	{attribute 'TcIecLibraryType'}
	{attribute 'external_name' := 'F_VN_InsertIntoContainer_TcVnRotatedRectangle_GUID_7CAC9217_ADAF_D1DF_8A4B_C5D37D5C5790'}
	(* Insert an element of type TcVnRotatedRectangle into a container before the specified position. *)
	FUNCTION F_VN_InsertIntoContainer_TcVnRotatedRectangle : HRESULT
	VAR_IN_OUT
		stElement	:	TcVnRotatedRectangle;	(* Single element to insert into ipContainer *)
	END_VAR
	VAR_INPUT
		ipContainer	:	ITcVnContainer;	(* Container in which to insert the element *)
		nIndex	:	ULINT;	(* Position, before which the element will be inserted *)
		hrPrev	:	HRESULT;	(* HRESULT indicating the result of previous operations (If SUCCEEDED(hrPrev) equals false, no operation is executed.) *)
	END_VAR

END_FUNCTION

// Functions/Basic Container Operations/F_VN_InsertIntoContainer/F_VN_InsertIntoContainer_TcVnVector2_DINT

	{attribute 'TcIecLibraryType'}
	{attribute 'external_name' := 'F_VN_InsertIntoContainer_TcVnVector2_DINT_GUID_6566CC88_DAB0_D931_BB59_6B341F06AF09'}
	(* Insert an element of type TcVnVector2_DINT into a container before the specified position. *)
	FUNCTION F_VN_InsertIntoContainer_TcVnVector2_DINT : HRESULT
	VAR_IN_OUT
		aElement	:	TcVnVector2_DINT;	(* Single element to insert into ipContainer *)
	END_VAR
	VAR_INPUT
		ipContainer	:	ITcVnContainer;	(* Container in which to insert the element *)
		nIndex	:	ULINT;	(* Position, before which the element will be inserted *)
		hrPrev	:	HRESULT;	(* HRESULT indicating the result of previous operations (If SUCCEEDED(hrPrev) equals false, no operation is executed.) *)
	END_VAR

END_FUNCTION

// Functions/Basic Container Operations/F_VN_InsertIntoContainer/F_VN_InsertIntoContainer_TcVnVector2_INT

	{attribute 'TcIecLibraryType'}
	{attribute 'external_name' := 'F_VN_InsertIntoContainer_TcVnVector2_INT_GUID_1A44D456_0A40_D7BF_84B8_D447168CEA63'}
	(* Insert an element of type TcVnVector2_INT into a container before the specified position. *)
	FUNCTION F_VN_InsertIntoContainer_TcVnVector2_INT : HRESULT
	VAR_IN_OUT
		aElement	:	TcVnVector2_INT;	(* Single element to insert into ipContainer *)
	END_VAR
	VAR_INPUT
		ipContainer	:	ITcVnContainer;	(* Container in which to insert the element *)
		nIndex	:	ULINT;	(* Position, before which the element will be inserted *)
		hrPrev	:	HRESULT;	(* HRESULT indicating the result of previous operations (If SUCCEEDED(hrPrev) equals false, no operation is executed.) *)
	END_VAR

END_FUNCTION

// Functions/Basic Container Operations/F_VN_InsertIntoContainer/F_VN_InsertIntoContainer_TcVnVector2_REAL

	{attribute 'TcIecLibraryType'}
	{attribute 'external_name' := 'F_VN_InsertIntoContainer_TcVnVector2_REAL_GUID_14F4E4FE_449B_DEBB_AC09_B5A9FB146C7C'}
	(* Insert an element of type TcVnVector2_REAL into a container before the specified position. *)
	FUNCTION F_VN_InsertIntoContainer_TcVnVector2_REAL : HRESULT
	VAR_IN_OUT
		aElement	:	TcVnVector2_REAL;	(* Single element to insert into ipContainer *)
	END_VAR
	VAR_INPUT
		ipContainer	:	ITcVnContainer;	(* Container in which to insert the element *)
		nIndex	:	ULINT;	(* Position, before which the element will be inserted *)
		hrPrev	:	HRESULT;	(* HRESULT indicating the result of previous operations (If SUCCEEDED(hrPrev) equals false, no operation is executed.) *)
	END_VAR

END_FUNCTION

// Functions/Basic Container Operations/F_VN_InsertIntoContainer/F_VN_InsertIntoContainer_TcVnVector2_SINT

	{attribute 'TcIecLibraryType'}
	{attribute 'external_name' := 'F_VN_InsertIntoContainer_TcVnVector2_SINT_GUID_4FA6BDE4_FC4B_D14F_9AAD_DECDAC1A2485'}
	(* Insert an element of type TcVnVector2_SINT into a container before the specified position. *)
	FUNCTION F_VN_InsertIntoContainer_TcVnVector2_SINT : HRESULT
	VAR_IN_OUT
		aElement	:	TcVnVector2_SINT;	(* Single element to insert into ipContainer *)
	END_VAR
	VAR_INPUT
		ipContainer	:	ITcVnContainer;	(* Container in which to insert the element *)
		nIndex	:	ULINT;	(* Position, before which the element will be inserted *)
		hrPrev	:	HRESULT;	(* HRESULT indicating the result of previous operations (If SUCCEEDED(hrPrev) equals false, no operation is executed.) *)
	END_VAR

END_FUNCTION

// Functions/Basic Container Operations/F_VN_InsertIntoContainer/F_VN_InsertIntoContainer_TcVnVector2_UINT

	{attribute 'TcIecLibraryType'}
	{attribute 'external_name' := 'F_VN_InsertIntoContainer_TcVnVector2_UINT_GUID_EB7FA824_1233_DA1F_B08D_37FDC60F70A2'}
	(* Insert an element of type TcVnVector2_UINT into a container before the specified position. *)
	FUNCTION F_VN_InsertIntoContainer_TcVnVector2_UINT : HRESULT
	VAR_IN_OUT
		aElement	:	TcVnVector2_UINT;	(* Single element to insert into ipContainer *)
	END_VAR
	VAR_INPUT
		ipContainer	:	ITcVnContainer;	(* Container in which to insert the element *)
		nIndex	:	ULINT;	(* Position, before which the element will be inserted *)
		hrPrev	:	HRESULT;	(* HRESULT indicating the result of previous operations (If SUCCEEDED(hrPrev) equals false, no operation is executed.) *)
	END_VAR

END_FUNCTION

// Functions/Basic Container Operations/F_VN_InsertIntoContainer/F_VN_InsertIntoContainer_TcVnVector2_USINT

	{attribute 'TcIecLibraryType'}
	{attribute 'external_name' := 'F_VN_InsertIntoContainer_TcVnVector2_USINT_GUID_68AD2749_FA5E_D5AF_8F19_582165BB6F3C'}
	(* Insert an element of type TcVnVector2_USINT into a container before the specified position. *)
	FUNCTION F_VN_InsertIntoContainer_TcVnVector2_USINT : HRESULT
	VAR_IN_OUT
		aElement	:	TcVnVector2_USINT;	(* Single element to insert into ipContainer *)
	END_VAR
	VAR_INPUT
		ipContainer	:	ITcVnContainer;	(* Container in which to insert the element *)
		nIndex	:	ULINT;	(* Position, before which the element will be inserted *)
		hrPrev	:	HRESULT;	(* HRESULT indicating the result of previous operations (If SUCCEEDED(hrPrev) equals false, no operation is executed.) *)
	END_VAR

END_FUNCTION

// Functions/Basic Container Operations/F_VN_InsertIntoContainer/F_VN_InsertIntoContainer_TcVnVector3_INT

	{attribute 'TcIecLibraryType'}
	{attribute 'external_name' := 'F_VN_InsertIntoContainer_TcVnVector3_INT_GUID_A6543EEA_C009_D51F_BEE7_FF579A0CBCDE'}
	(* Insert an element of type TcVnVector3_INT into a container before the specified position. *)
	FUNCTION F_VN_InsertIntoContainer_TcVnVector3_INT : HRESULT
	VAR_IN_OUT
		aElement	:	TcVnVector3_INT;	(* Single element to insert into ipContainer *)
	END_VAR
	VAR_INPUT
		ipContainer	:	ITcVnContainer;	(* Container in which to insert the element *)
		nIndex	:	ULINT;	(* Position, before which the element will be inserted *)
		hrPrev	:	HRESULT;	(* HRESULT indicating the result of previous operations (If SUCCEEDED(hrPrev) equals false, no operation is executed.) *)
	END_VAR

END_FUNCTION

// Functions/Basic Container Operations/F_VN_InsertIntoContainer/F_VN_InsertIntoContainer_TcVnVector3_REAL

	{attribute 'TcIecLibraryType'}
	{attribute 'external_name' := 'F_VN_InsertIntoContainer_TcVnVector3_REAL_GUID_8DA4CB93_E662_DD0B_B77C_47E33715929C'}
	(* Insert an element of type TcVnVector3_REAL into a container before the specified position. *)
	FUNCTION F_VN_InsertIntoContainer_TcVnVector3_REAL : HRESULT
	VAR_IN_OUT
		aElement	:	TcVnVector3_REAL;	(* Single element to insert into ipContainer *)
	END_VAR
	VAR_INPUT
		ipContainer	:	ITcVnContainer;	(* Container in which to insert the element *)
		nIndex	:	ULINT;	(* Position, before which the element will be inserted *)
		hrPrev	:	HRESULT;	(* HRESULT indicating the result of previous operations (If SUCCEEDED(hrPrev) equals false, no operation is executed.) *)
	END_VAR

END_FUNCTION

// Functions/Basic Container Operations/F_VN_InsertIntoContainer/F_VN_InsertIntoContainer_TcVnVector3_SINT

	{attribute 'TcIecLibraryType'}
	{attribute 'external_name' := 'F_VN_InsertIntoContainer_TcVnVector3_SINT_GUID_9F083386_9C91_DC08_8219_0E1B3C149953'}
	(* Insert an element of type TcVnVector3_SINT into a container before the specified position. *)
	FUNCTION F_VN_InsertIntoContainer_TcVnVector3_SINT : HRESULT
	VAR_IN_OUT
		aElement	:	TcVnVector3_SINT;	(* Single element to insert into ipContainer *)
	END_VAR
	VAR_INPUT
		ipContainer	:	ITcVnContainer;	(* Container in which to insert the element *)
		nIndex	:	ULINT;	(* Position, before which the element will be inserted *)
		hrPrev	:	HRESULT;	(* HRESULT indicating the result of previous operations (If SUCCEEDED(hrPrev) equals false, no operation is executed.) *)
	END_VAR

END_FUNCTION

// Functions/Basic Container Operations/F_VN_InsertIntoContainer/F_VN_InsertIntoContainer_TcVnVector3_UINT

	{attribute 'TcIecLibraryType'}
	{attribute 'external_name' := 'F_VN_InsertIntoContainer_TcVnVector3_UINT_GUID_A8405EB2_25DD_DB35_B4DF_AFF6C48501DC'}
	(* Insert an element of type TcVnVector3_UINT into a container before the specified position. *)
	FUNCTION F_VN_InsertIntoContainer_TcVnVector3_UINT : HRESULT
	VAR_IN_OUT
		aElement	:	TcVnVector3_UINT;	(* Single element to insert into ipContainer *)
	END_VAR
	VAR_INPUT
		ipContainer	:	ITcVnContainer;	(* Container in which to insert the element *)
		nIndex	:	ULINT;	(* Position, before which the element will be inserted *)
		hrPrev	:	HRESULT;	(* HRESULT indicating the result of previous operations (If SUCCEEDED(hrPrev) equals false, no operation is executed.) *)
	END_VAR

END_FUNCTION

// Functions/Basic Container Operations/F_VN_InsertIntoContainer/F_VN_InsertIntoContainer_TcVnVector3_USINT

	{attribute 'TcIecLibraryType'}
	{attribute 'external_name' := 'F_VN_InsertIntoContainer_TcVnVector3_USINT_GUID_C1142200_49EE_D153_9630_C3BAFAFB5C22'}
	(* Insert an element of type TcVnVector3_USINT into a container before the specified position. *)
	FUNCTION F_VN_InsertIntoContainer_TcVnVector3_USINT : HRESULT
	VAR_IN_OUT
		aElement	:	TcVnVector3_USINT;	(* Single element to insert into ipContainer *)
	END_VAR
	VAR_INPUT
		ipContainer	:	ITcVnContainer;	(* Container in which to insert the element *)
		nIndex	:	ULINT;	(* Position, before which the element will be inserted *)
		hrPrev	:	HRESULT;	(* HRESULT indicating the result of previous operations (If SUCCEEDED(hrPrev) equals false, no operation is executed.) *)
	END_VAR

END_FUNCTION

// Functions/Basic Container Operations/F_VN_InsertIntoContainer/F_VN_InsertIntoContainer_TcVnVector4_DINT

	{attribute 'TcIecLibraryType'}
	{attribute 'external_name' := 'F_VN_InsertIntoContainer_TcVnVector4_DINT_GUID_B98F2330_DD6A_D95D_8783_2B0449E0CC84'}
	(* Insert an element of type TcVnVector4_DINT into a container before the specified position. *)
	FUNCTION F_VN_InsertIntoContainer_TcVnVector4_DINT : HRESULT
	VAR_IN_OUT
		aElement	:	TcVnVector4_DINT;	(* Single element to insert into ipContainer *)
	END_VAR
	VAR_INPUT
		ipContainer	:	ITcVnContainer;	(* Container in which to insert the element *)
		nIndex	:	ULINT;	(* Position, before which the element will be inserted *)
		hrPrev	:	HRESULT;	(* HRESULT indicating the result of previous operations (If SUCCEEDED(hrPrev) equals false, no operation is executed.) *)
	END_VAR

END_FUNCTION

// Functions/Basic Container Operations/F_VN_InsertIntoContainer/F_VN_InsertIntoContainer_TcVnVector4_INT

	{attribute 'TcIecLibraryType'}
	{attribute 'external_name' := 'F_VN_InsertIntoContainer_TcVnVector4_INT_GUID_65611BB7_30D8_D8ED_8ECE_E86DF68481D6'}
	(* Insert an element of type TcVnVector4_INT into a container before the specified position. *)
	FUNCTION F_VN_InsertIntoContainer_TcVnVector4_INT : HRESULT
	VAR_IN_OUT
		aElement	:	TcVnVector4_INT;	(* Single element to insert into ipContainer *)
	END_VAR
	VAR_INPUT
		ipContainer	:	ITcVnContainer;	(* Container in which to insert the element *)
		nIndex	:	ULINT;	(* Position, before which the element will be inserted *)
		hrPrev	:	HRESULT;	(* HRESULT indicating the result of previous operations (If SUCCEEDED(hrPrev) equals false, no operation is executed.) *)
	END_VAR

END_FUNCTION

// Functions/Basic Container Operations/F_VN_InsertIntoContainer/F_VN_InsertIntoContainer_TcVnVector4_LREAL

	{attribute 'TcIecLibraryType'}
	{attribute 'external_name' := 'F_VN_InsertIntoContainer_TcVnVector4_LREAL_GUID_FE564EF4_0166_DE95_B96B_4103EC79B71E'}
	(* Insert an element of type TcVnVector4_LREAL into a container before the specified position. *)
	FUNCTION F_VN_InsertIntoContainer_TcVnVector4_LREAL : HRESULT
	VAR_IN_OUT
		aElement	:	TcVnVector4_LREAL;	(* Single element to insert into ipContainer *)
	END_VAR
	VAR_INPUT
		ipContainer	:	ITcVnContainer;	(* Container in which to insert the element *)
		nIndex	:	ULINT;	(* Position, before which the element will be inserted *)
		hrPrev	:	HRESULT;	(* HRESULT indicating the result of previous operations (If SUCCEEDED(hrPrev) equals false, no operation is executed.) *)
	END_VAR

END_FUNCTION

// Functions/Basic Container Operations/F_VN_InsertIntoContainer/F_VN_InsertIntoContainer_TcVnVector4_REAL

	{attribute 'TcIecLibraryType'}
	{attribute 'external_name' := 'F_VN_InsertIntoContainer_TcVnVector4_REAL_GUID_58C4540D_8F55_DF4C_9020_215109A1688E'}
	(* Insert an element of type TcVnVector4_REAL into a container before the specified position. *)
	FUNCTION F_VN_InsertIntoContainer_TcVnVector4_REAL : HRESULT
	VAR_IN_OUT
		aElement	:	TcVnVector4_REAL;	(* Single element to insert into ipContainer *)
	END_VAR
	VAR_INPUT
		ipContainer	:	ITcVnContainer;	(* Container in which to insert the element *)
		nIndex	:	ULINT;	(* Position, before which the element will be inserted *)
		hrPrev	:	HRESULT;	(* HRESULT indicating the result of previous operations (If SUCCEEDED(hrPrev) equals false, no operation is executed.) *)
	END_VAR

END_FUNCTION

// Functions/Basic Container Operations/F_VN_InsertIntoContainer/F_VN_InsertIntoContainer_TcVnVector4_SINT

	{attribute 'TcIecLibraryType'}
	{attribute 'external_name' := 'F_VN_InsertIntoContainer_TcVnVector4_SINT_GUID_E59FA623_EBB2_DB93_9AF8_202896EF00E4'}
	(* Insert an element of type TcVnVector4_SINT into a container before the specified position. *)
	FUNCTION F_VN_InsertIntoContainer_TcVnVector4_SINT : HRESULT
	VAR_IN_OUT
		aElement	:	TcVnVector4_SINT;	(* Single element to insert into ipContainer *)
	END_VAR
	VAR_INPUT
		ipContainer	:	ITcVnContainer;	(* Container in which to insert the element *)
		nIndex	:	ULINT;	(* Position, before which the element will be inserted *)
		hrPrev	:	HRESULT;	(* HRESULT indicating the result of previous operations (If SUCCEEDED(hrPrev) equals false, no operation is executed.) *)
	END_VAR

END_FUNCTION

// Functions/Basic Container Operations/F_VN_InsertIntoContainer/F_VN_InsertIntoContainer_TcVnVector4_UINT

	{attribute 'TcIecLibraryType'}
	{attribute 'external_name' := 'F_VN_InsertIntoContainer_TcVnVector4_UINT_GUID_52ADF8A2_FEB4_DF8A_9994_E3F816D9D014'}
	(* Insert an element of type TcVnVector4_UINT into a container before the specified position. *)
	FUNCTION F_VN_InsertIntoContainer_TcVnVector4_UINT : HRESULT
	VAR_IN_OUT
		aElement	:	TcVnVector4_UINT;	(* Single element to insert into ipContainer *)
	END_VAR
	VAR_INPUT
		ipContainer	:	ITcVnContainer;	(* Container in which to insert the element *)
		nIndex	:	ULINT;	(* Position, before which the element will be inserted *)
		hrPrev	:	HRESULT;	(* HRESULT indicating the result of previous operations (If SUCCEEDED(hrPrev) equals false, no operation is executed.) *)
	END_VAR

END_FUNCTION

// Functions/Basic Container Operations/F_VN_InsertIntoContainer/F_VN_InsertIntoContainer_TcVnVector4_USINT

	{attribute 'TcIecLibraryType'}
	{attribute 'external_name' := 'F_VN_InsertIntoContainer_TcVnVector4_USINT_GUID_8D180FCF_4F7F_D25B_9D06_29434C4138AE'}
	(* Insert an element of type TcVnVector4_USINT into a container before the specified position. *)
	FUNCTION F_VN_InsertIntoContainer_TcVnVector4_USINT : HRESULT
	VAR_IN_OUT
		aElement	:	TcVnVector4_USINT;	(* Single element to insert into ipContainer *)
	END_VAR
	VAR_INPUT
		ipContainer	:	ITcVnContainer;	(* Container in which to insert the element *)
		nIndex	:	ULINT;	(* Position, before which the element will be inserted *)
		hrPrev	:	HRESULT;	(* HRESULT indicating the result of previous operations (If SUCCEEDED(hrPrev) equals false, no operation is executed.) *)
	END_VAR

END_FUNCTION

// Functions/Basic Container Operations/F_VN_InsertIntoContainer/F_VN_InsertIntoContainer_UDINT

	{attribute 'TcIecLibraryType'}
	{attribute 'external_name' := 'F_VN_InsertIntoContainer_UDINT_GUID_456412AD_2528_D507_8741_196A0EE9AFE2'}
	(* Insert an element of type UDINT into a container before the specified position. *)
	FUNCTION F_VN_InsertIntoContainer_UDINT : HRESULT
	VAR_INPUT
		nElement	:	UDINT;	(* Single element to insert into ipContainer *)
		ipContainer	:	ITcVnContainer;	(* Container in which to insert the element *)
		nIndex	:	ULINT;	(* Position, before which the element will be inserted *)
		hrPrev	:	HRESULT;	(* HRESULT indicating the result of previous operations (If SUCCEEDED(hrPrev) equals false, no operation is executed.) *)
	END_VAR

END_FUNCTION

// Functions/Basic Container Operations/F_VN_InsertIntoContainer/F_VN_InsertIntoContainer_UINT

	{attribute 'TcIecLibraryType'}
	{attribute 'external_name' := 'F_VN_InsertIntoContainer_UINT_GUID_6B49D457_9F4E_DE5F_85EF_D3413FF89161'}
	(* Insert an element of type UINT into a container before the specified position. *)
	FUNCTION F_VN_InsertIntoContainer_UINT : HRESULT
	VAR_INPUT
		nElement	:	UINT;	(* Single element to insert into ipContainer *)
		ipContainer	:	ITcVnContainer;	(* Container in which to insert the element *)
		nIndex	:	ULINT;	(* Position, before which the element will be inserted *)
		hrPrev	:	HRESULT;	(* HRESULT indicating the result of previous operations (If SUCCEEDED(hrPrev) equals false, no operation is executed.) *)
	END_VAR

END_FUNCTION

// Functions/Basic Container Operations/F_VN_InsertIntoContainer/F_VN_InsertIntoContainer_ULINT

	{attribute 'TcIecLibraryType'}
	{attribute 'external_name' := 'F_VN_InsertIntoContainer_ULINT_GUID_FE1D7BC2_89AC_D4A6_855E_4E891AD80812'}
	(* Insert an element of type ULINT into a container before the specified position. *)
	FUNCTION F_VN_InsertIntoContainer_ULINT : HRESULT
	VAR_INPUT
		nElement	:	ULINT;	(* Single element to insert into ipContainer *)
		ipContainer	:	ITcVnContainer;	(* Container in which to insert the element *)
		nIndex	:	ULINT;	(* Position, before which the element will be inserted *)
		hrPrev	:	HRESULT;	(* HRESULT indicating the result of previous operations (If SUCCEEDED(hrPrev) equals false, no operation is executed.) *)
	END_VAR

END_FUNCTION

// Functions/Basic Container Operations/F_VN_InsertIntoContainer/F_VN_InsertIntoContainer_USINT

	{attribute 'TcIecLibraryType'}
	{attribute 'external_name' := 'F_VN_InsertIntoContainer_USINT_GUID_A85F087B_469C_DB69_A492_76C66B672E9A'}
	(* Insert an element of type USINT into a container before the specified position. *)
	FUNCTION F_VN_InsertIntoContainer_USINT : HRESULT
	VAR_INPUT
		nElement	:	USINT;	(* Single element to insert into ipContainer *)
		ipContainer	:	ITcVnContainer;	(* Container in which to insert the element *)
		nIndex	:	ULINT;	(* Position, before which the element will be inserted *)
		hrPrev	:	HRESULT;	(* HRESULT indicating the result of previous operations (If SUCCEEDED(hrPrev) equals false, no operation is executed.) *)
	END_VAR

END_FUNCTION

// Functions/Basic Container Operations/F_VN_SetAt/F_VN_SetAt_ITcVnContainer

	{attribute 'TcIecLibraryType'}
	{attribute 'external_name' := 'F_VN_SetAt_ITcVnContainer_GUID_B4D766E9_0AA2_DD2D_B478_52D12AAD3DA2'}
	(* Sets the element at the specified index of the container. (Alternatively use interface method .SetAt.) *)
	FUNCTION F_VN_SetAt_ITcVnContainer : HRESULT
	VAR_INPUT
		ipElement	:	ITcVnContainer;	(* Element to set at the specified container position *)
		ipContainer	:	ITcVnContainer;	(* Container with ITcVnContainer elements, in which the element at position nIndex is replaced by ipElement *)
		nIndex	:	ULINT;	(* Index *)
		hrPrev	:	HRESULT;	(* HRESULT indicating the result of previous operations (If SUCCEEDED(hrPrev) equals false, no operation is executed.) *)
	END_VAR

END_FUNCTION

// Functions/Basic Container Operations/F_VN_SetAt/F_VN_SetAt_DINT

	{attribute 'TcIecLibraryType'}
	{attribute 'external_name' := 'F_VN_SetAt_DINT_GUID_253433CB_2425_DDF0_8BE6_B05C6CBF2EB5'}
	(* Sets the element at the specified index of the container. *)
	FUNCTION F_VN_SetAt_DINT : HRESULT
	VAR_INPUT
		nElement	:	DINT;	(* Element to set at the specified container position *)
		ipContainer	:	ITcVnContainer;	(* Container with DINT elements, in which the element at position nIndex is replaced by nElement *)
		nIndex	:	ULINT;	(* Index *)
		hrPrev	:	HRESULT;	(* HRESULT indicating the result of previous operations (If SUCCEEDED(hrPrev) equals false, no operation is executed.) *)
	END_VAR

END_FUNCTION

// Functions/Basic Container Operations/F_VN_SetAt/F_VN_SetAt_INT

	{attribute 'TcIecLibraryType'}
	{attribute 'external_name' := 'F_VN_SetAt_INT_GUID_B0E2F6D5_1415_D22F_A65C_C36499F3DF8D'}
	(* Sets the element at the specified index of the container. *)
	FUNCTION F_VN_SetAt_INT : HRESULT
	VAR_INPUT
		nElement	:	INT;	(* Element to set at the specified container position *)
		ipContainer	:	ITcVnContainer;	(* Container with INT elements, in which the element at position nIndex is replaced by nElement *)
		nIndex	:	ULINT;	(* Index *)
		hrPrev	:	HRESULT;	(* HRESULT indicating the result of previous operations (If SUCCEEDED(hrPrev) equals false, no operation is executed.) *)
	END_VAR

END_FUNCTION

// Functions/Basic Container Operations/F_VN_SetAt/F_VN_SetAt_ITcVnImage

	{attribute 'TcIecLibraryType'}
	{attribute 'external_name' := 'F_VN_SetAt_ITcVnImage_GUID_8BFD8EA5_9C85_DADE_A61A_698800738790'}
	(* Sets the element at the specified index of the container. *)
	FUNCTION F_VN_SetAt_ITcVnImage : HRESULT
	VAR_INPUT
		ipElement	:	ITcVnImage;	(* Element to set at the specified container position *)
		ipContainer	:	ITcVnContainer;	(* Container with ITcVnImage elements, in which the element at position nIndex is replaced by ipElement *)
		nIndex	:	ULINT;	(* Index *)
		hrPrev	:	HRESULT;	(* HRESULT indicating the result of previous operations (If SUCCEEDED(hrPrev) equals false, no operation is executed.) *)
	END_VAR

END_FUNCTION

// Functions/Basic Container Operations/F_VN_SetAt/F_VN_SetAt_LREAL

	{attribute 'TcIecLibraryType'}
	{attribute 'external_name' := 'F_VN_SetAt_LREAL_GUID_B183A29F_8335_D912_8808_5352ACF3B9D5'}
	(* Sets the element at the specified index of the container. *)
	FUNCTION F_VN_SetAt_LREAL : HRESULT
	VAR_INPUT
		fElement	:	LREAL;	(* Element to set at the specified container position *)
		ipContainer	:	ITcVnContainer;	(* Container with LREAL elements, in which the element at position nIndex is replaced by fElement *)
		nIndex	:	ULINT;	(* Index *)
		hrPrev	:	HRESULT;	(* HRESULT indicating the result of previous operations (If SUCCEEDED(hrPrev) equals false, no operation is executed.) *)
	END_VAR

END_FUNCTION

// Functions/Basic Container Operations/F_VN_SetAt/F_VN_SetAt_REAL

	{attribute 'TcIecLibraryType'}
	{attribute 'external_name' := 'F_VN_SetAt_REAL_GUID_7E957C6A_9FEC_D57C_9D71_8DD5085B7449'}
	(* Sets the element at the specified index of the container. *)
	FUNCTION F_VN_SetAt_REAL : HRESULT
	VAR_INPUT
		fElement	:	REAL;	(* Element to set at the specified container position *)
		ipContainer	:	ITcVnContainer;	(* Container with REAL elements, in which the element at position nIndex is replaced by fElement *)
		nIndex	:	ULINT;	(* Index *)
		hrPrev	:	HRESULT;	(* HRESULT indicating the result of previous operations (If SUCCEEDED(hrPrev) equals false, no operation is executed.) *)
	END_VAR

END_FUNCTION

// Functions/Basic Container Operations/F_VN_SetAt/F_VN_SetAt_SINT

	{attribute 'TcIecLibraryType'}
	{attribute 'external_name' := 'F_VN_SetAt_SINT_GUID_A0498278_0B8F_D4D0_B592_136B0477C0F3'}
	(* Sets the element at the specified index of the container. *)
	FUNCTION F_VN_SetAt_SINT : HRESULT
	VAR_INPUT
		nElement	:	SINT;	(* Element to set at the specified container position *)
		ipContainer	:	ITcVnContainer;	(* Container with SINT elements, in which the element at position nIndex is replaced by nElement *)
		nIndex	:	ULINT;	(* Index *)
		hrPrev	:	HRESULT;	(* HRESULT indicating the result of previous operations (If SUCCEEDED(hrPrev) equals false, no operation is executed.) *)
	END_VAR

END_FUNCTION

// Functions/Basic Container Operations/F_VN_SetAt/F_VN_SetAt_TcVnDMatch

	{attribute 'TcIecLibraryType'}
	{attribute 'external_name' := 'F_VN_SetAt_TcVnDMatch_GUID_2DD68088_896B_D3C6_AD71_4673DA0389D4'}
	(* Sets the element at the specified index of the container. *)
	FUNCTION F_VN_SetAt_TcVnDMatch : HRESULT
	VAR_IN_OUT
		stElement	:	TcVnDMatch;	(* Element to set at the specified container position *)
	END_VAR
	VAR_INPUT
		ipContainer	:	ITcVnContainer;	(* Container with TcVnDMatch elements, in which the element at position nIndex is replaced by stElement *)
		nIndex	:	ULINT;	(* Index *)
		hrPrev	:	HRESULT;	(* HRESULT indicating the result of previous operations (If SUCCEEDED(hrPrev) equals false, no operation is executed.) *)
	END_VAR

END_FUNCTION

// Functions/Basic Container Operations/F_VN_SetAt/F_VN_SetAt_TcVnKeyPoint

	{attribute 'TcIecLibraryType'}
	{attribute 'external_name' := 'F_VN_SetAt_TcVnKeyPoint_GUID_5542B220_7839_DF8E_B6D3_14C96E222448'}
	(* Sets the element at the specified index of the container. *)
	FUNCTION F_VN_SetAt_TcVnKeyPoint : HRESULT
	VAR_IN_OUT
		stElement	:	TcVnKeyPoint;	(* Element to set at the specified container position *)
	END_VAR
	VAR_INPUT
		ipContainer	:	ITcVnContainer;	(* Container with TcVnKeyPoint elements, in which the element at position nIndex is replaced by stElement *)
		nIndex	:	ULINT;	(* Index *)
		hrPrev	:	HRESULT;	(* HRESULT indicating the result of previous operations (If SUCCEEDED(hrPrev) equals false, no operation is executed.) *)
	END_VAR

END_FUNCTION

// Functions/Basic Container Operations/F_VN_SetAt/F_VN_SetAt_TcVnPoint2_DINT

	{attribute 'TcIecLibraryType'}
	{attribute 'external_name' := 'F_VN_SetAt_TcVnPoint2_DINT_GUID_380C3A28_A538_D35A_886E_4DB239484DC0'}
	(* Sets the element at the specified index of the container. *)
	FUNCTION F_VN_SetAt_TcVnPoint2_DINT : HRESULT
	VAR_IN_OUT
		aElement	:	TcVnPoint2_DINT;	(* Element to set at the specified container position *)
	END_VAR
	VAR_INPUT
		ipContainer	:	ITcVnContainer;	(* Container with TcVnPoint2_DINT elements, in which the element at position nIndex is replaced by aElement *)
		nIndex	:	ULINT;	(* Index *)
		hrPrev	:	HRESULT;	(* HRESULT indicating the result of previous operations (If SUCCEEDED(hrPrev) equals false, no operation is executed.) *)
	END_VAR

END_FUNCTION

// Functions/Basic Container Operations/F_VN_SetAt/F_VN_SetAt_TcVnPoint2_LREAL

	{attribute 'TcIecLibraryType'}
	{attribute 'external_name' := 'F_VN_SetAt_TcVnPoint2_LREAL_GUID_3335CF1D_E3D4_D03B_9014_F1A43D08A30F'}
	(* Sets the element at the specified index of the container. *)
	FUNCTION F_VN_SetAt_TcVnPoint2_LREAL : HRESULT
	VAR_IN_OUT
		aElement	:	TcVnPoint2_LREAL;	(* Element to set at the specified container position *)
	END_VAR
	VAR_INPUT
		ipContainer	:	ITcVnContainer;	(* Container with TcVnPoint2_LREAL elements, in which the element at position nIndex is replaced by aElement *)
		nIndex	:	ULINT;	(* Index *)
		hrPrev	:	HRESULT;	(* HRESULT indicating the result of previous operations (If SUCCEEDED(hrPrev) equals false, no operation is executed.) *)
	END_VAR

END_FUNCTION

// Functions/Basic Container Operations/F_VN_SetAt/F_VN_SetAt_TcVnPoint2_REAL

	{attribute 'TcIecLibraryType'}
	{attribute 'external_name' := 'F_VN_SetAt_TcVnPoint2_REAL_GUID_633C5783_5133_DC7E_ABCC_93BD16D56EFF'}
	(* Sets the element at the specified index of the container. *)
	FUNCTION F_VN_SetAt_TcVnPoint2_REAL : HRESULT
	VAR_IN_OUT
		aElement	:	TcVnPoint2_REAL;	(* Element to set at the specified container position *)
	END_VAR
	VAR_INPUT
		ipContainer	:	ITcVnContainer;	(* Container with TcVnPoint2_REAL elements, in which the element at position nIndex is replaced by aElement *)
		nIndex	:	ULINT;	(* Index *)
		hrPrev	:	HRESULT;	(* HRESULT indicating the result of previous operations (If SUCCEEDED(hrPrev) equals false, no operation is executed.) *)
	END_VAR

END_FUNCTION

// Functions/Basic Container Operations/F_VN_SetAt/F_VN_SetAt_TcVnPoint3_LREAL

	{attribute 'TcIecLibraryType'}
	{attribute 'external_name' := 'F_VN_SetAt_TcVnPoint3_LREAL_GUID_FA067292_14A4_D164_A359_A281C2761513'}
	(* Sets the element at the specified index of the container. *)
	FUNCTION F_VN_SetAt_TcVnPoint3_LREAL : HRESULT
	VAR_IN_OUT
		aElement	:	TcVnPoint3_LREAL;	(* Element to set at the specified container position *)
	END_VAR
	VAR_INPUT
		ipContainer	:	ITcVnContainer;	(* Container with TcVnPoint3_LREAL elements, in which the element at position nIndex is replaced by aElement *)
		nIndex	:	ULINT;	(* Index *)
		hrPrev	:	HRESULT;	(* HRESULT indicating the result of previous operations (If SUCCEEDED(hrPrev) equals false, no operation is executed.) *)
	END_VAR

END_FUNCTION

// Functions/Basic Container Operations/F_VN_SetAt/F_VN_SetAt_TcVnPoint3_REAL

	{attribute 'TcIecLibraryType'}
	{attribute 'external_name' := 'F_VN_SetAt_TcVnPoint3_REAL_GUID_C913190D_69EF_DE67_9951_6D3EB8AF0AD3'}
	(* Sets the element at the specified index of the container. *)
	FUNCTION F_VN_SetAt_TcVnPoint3_REAL : HRESULT
	VAR_IN_OUT
		aElement	:	TcVnPoint3_REAL;	(* Element to set at the specified container position *)
	END_VAR
	VAR_INPUT
		ipContainer	:	ITcVnContainer;	(* Container with TcVnPoint3_REAL elements, in which the element at position nIndex is replaced by aElement *)
		nIndex	:	ULINT;	(* Index *)
		hrPrev	:	HRESULT;	(* HRESULT indicating the result of previous operations (If SUCCEEDED(hrPrev) equals false, no operation is executed.) *)
	END_VAR

END_FUNCTION

// Functions/Basic Container Operations/F_VN_SetAt/F_VN_SetAt_TcVnRectangle_DINT

	{attribute 'TcIecLibraryType'}
	{attribute 'external_name' := 'F_VN_SetAt_TcVnRectangle_DINT_GUID_4532A8D1_EA7C_DA26_B932_400B95600032'}
	(* Sets the element at the specified index of the container. *)
	FUNCTION F_VN_SetAt_TcVnRectangle_DINT : HRESULT
	VAR_IN_OUT
		stElement	:	TcVnRectangle_DINT;	(* Element to set at the specified container position *)
	END_VAR
	VAR_INPUT
		ipContainer	:	ITcVnContainer;	(* Container with TcVnRectangle_DINT elements, in which the element at position nIndex is replaced by stElement *)
		nIndex	:	ULINT;	(* Index *)
		hrPrev	:	HRESULT;	(* HRESULT indicating the result of previous operations (If SUCCEEDED(hrPrev) equals false, no operation is executed.) *)
	END_VAR

END_FUNCTION

// Functions/Basic Container Operations/F_VN_SetAt/F_VN_SetAt_TcVnRotatedRectangle

	{attribute 'TcIecLibraryType'}
	{attribute 'external_name' := 'F_VN_SetAt_TcVnRotatedRectangle_GUID_DAFC69FA_D3C4_DF12_83F3_1F7CE1D06A87'}
	(* Sets the element at the specified index of the container. *)
	FUNCTION F_VN_SetAt_TcVnRotatedRectangle : HRESULT
	VAR_IN_OUT
		stElement	:	TcVnRotatedRectangle;	(* Element to set at the specified container position *)
	END_VAR
	VAR_INPUT
		ipContainer	:	ITcVnContainer;	(* Container with TcVnRotatedRectangle elements, in which the element at position nIndex is replaced by stElement *)
		nIndex	:	ULINT;	(* Index *)
		hrPrev	:	HRESULT;	(* HRESULT indicating the result of previous operations (If SUCCEEDED(hrPrev) equals false, no operation is executed.) *)
	END_VAR

END_FUNCTION

// Functions/Basic Container Operations/F_VN_SetAt/F_VN_SetAt_TcVnVector2_DINT

	{attribute 'TcIecLibraryType'}
	{attribute 'external_name' := 'F_VN_SetAt_TcVnVector2_DINT_GUID_2E9C4D9D_A279_D002_86E8_DAA9F02A0E05'}
	(* Sets the element at the specified index of the container. *)
	FUNCTION F_VN_SetAt_TcVnVector2_DINT : HRESULT
	VAR_IN_OUT
		aElement	:	TcVnVector2_DINT;	(* Element to set at the specified container position *)
	END_VAR
	VAR_INPUT
		ipContainer	:	ITcVnContainer;	(* Container with TcVnVector2_DINT elements, in which the element at position nIndex is replaced by aElement *)
		nIndex	:	ULINT;	(* Index *)
		hrPrev	:	HRESULT;	(* HRESULT indicating the result of previous operations (If SUCCEEDED(hrPrev) equals false, no operation is executed.) *)
	END_VAR

END_FUNCTION

// Functions/Basic Container Operations/F_VN_SetAt/F_VN_SetAt_TcVnVector2_INT

	{attribute 'TcIecLibraryType'}
	{attribute 'external_name' := 'F_VN_SetAt_TcVnVector2_INT_GUID_EACA2057_16BA_D239_9B9E_74E17D255685'}
	(* Sets the element at the specified index of the container. *)
	FUNCTION F_VN_SetAt_TcVnVector2_INT : HRESULT
	VAR_IN_OUT
		aElement	:	TcVnVector2_INT;	(* Element to set at the specified container position *)
	END_VAR
	VAR_INPUT
		ipContainer	:	ITcVnContainer;	(* Container with TcVnVector2_INT elements, in which the element at position nIndex is replaced by aElement *)
		nIndex	:	ULINT;	(* Index *)
		hrPrev	:	HRESULT;	(* HRESULT indicating the result of previous operations (If SUCCEEDED(hrPrev) equals false, no operation is executed.) *)
	END_VAR

END_FUNCTION

// Functions/Basic Container Operations/F_VN_SetAt/F_VN_SetAt_TcVnVector2_REAL

	{attribute 'TcIecLibraryType'}
	{attribute 'external_name' := 'F_VN_SetAt_TcVnVector2_REAL_GUID_FCEEF9F1_A95E_D6B4_82C2_0524AF8ED162'}
	(* Sets the element at the specified index of the container. *)
	FUNCTION F_VN_SetAt_TcVnVector2_REAL : HRESULT
	VAR_IN_OUT
		aElement	:	TcVnVector2_REAL;	(* Element to set at the specified container position *)
	END_VAR
	VAR_INPUT
		ipContainer	:	ITcVnContainer;	(* Container with TcVnVector2_REAL elements, in which the element at position nIndex is replaced by aElement *)
		nIndex	:	ULINT;	(* Index *)
		hrPrev	:	HRESULT;	(* HRESULT indicating the result of previous operations (If SUCCEEDED(hrPrev) equals false, no operation is executed.) *)
	END_VAR

END_FUNCTION

// Functions/Basic Container Operations/F_VN_SetAt/F_VN_SetAt_TcVnVector2_SINT

	{attribute 'TcIecLibraryType'}
	{attribute 'external_name' := 'F_VN_SetAt_TcVnVector2_SINT_GUID_317C493E_1B6C_DEE3_AE25_CC2C29021A66'}
	(* Sets the element at the specified index of the container. *)
	FUNCTION F_VN_SetAt_TcVnVector2_SINT : HRESULT
	VAR_IN_OUT
		aElement	:	TcVnVector2_SINT;	(* Element to set at the specified container position *)
	END_VAR
	VAR_INPUT
		ipContainer	:	ITcVnContainer;	(* Container with TcVnVector2_SINT elements, in which the element at position nIndex is replaced by aElement *)
		nIndex	:	ULINT;	(* Index *)
		hrPrev	:	HRESULT;	(* HRESULT indicating the result of previous operations (If SUCCEEDED(hrPrev) equals false, no operation is executed.) *)
	END_VAR

END_FUNCTION

// Functions/Basic Container Operations/F_VN_SetAt/F_VN_SetAt_TcVnVector2_UINT

	{attribute 'TcIecLibraryType'}
	{attribute 'external_name' := 'F_VN_SetAt_TcVnVector2_UINT_GUID_51607B5B_B463_D36D_8B37_1F9AE2FB26C1'}
	(* Sets the element at the specified index of the container. *)
	FUNCTION F_VN_SetAt_TcVnVector2_UINT : HRESULT
	VAR_IN_OUT
		aElement	:	TcVnVector2_UINT;	(* Element to set at the specified container position *)
	END_VAR
	VAR_INPUT
		ipContainer	:	ITcVnContainer;	(* Container with TcVnVector2_UINT elements, in which the element at position nIndex is replaced by aElement *)
		nIndex	:	ULINT;	(* Index *)
		hrPrev	:	HRESULT;	(* HRESULT indicating the result of previous operations (If SUCCEEDED(hrPrev) equals false, no operation is executed.) *)
	END_VAR

END_FUNCTION

// Functions/Basic Container Operations/F_VN_SetAt/F_VN_SetAt_TcVnVector2_USINT

	{attribute 'TcIecLibraryType'}
	{attribute 'external_name' := 'F_VN_SetAt_TcVnVector2_USINT_GUID_01F9C5AE_E454_D0D0_90FA_2E0A2E622C7C'}
	(* Sets the element at the specified index of the container. *)
	FUNCTION F_VN_SetAt_TcVnVector2_USINT : HRESULT
	VAR_IN_OUT
		aElement	:	TcVnVector2_USINT;	(* Element to set at the specified container position *)
	END_VAR
	VAR_INPUT
		ipContainer	:	ITcVnContainer;	(* Container with TcVnVector2_USINT elements, in which the element at position nIndex is replaced by aElement *)
		nIndex	:	ULINT;	(* Index *)
		hrPrev	:	HRESULT;	(* HRESULT indicating the result of previous operations (If SUCCEEDED(hrPrev) equals false, no operation is executed.) *)
	END_VAR

END_FUNCTION

// Functions/Basic Container Operations/F_VN_SetAt/F_VN_SetAt_TcVnVector3_INT

	{attribute 'TcIecLibraryType'}
	{attribute 'external_name' := 'F_VN_SetAt_TcVnVector3_INT_GUID_C31915F3_E342_D7E4_A41C_3483F9896BDE'}
	(* Sets the element at the specified index of the container. *)
	FUNCTION F_VN_SetAt_TcVnVector3_INT : HRESULT
	VAR_IN_OUT
		aElement	:	TcVnVector3_INT;	(* Element to set at the specified container position *)
	END_VAR
	VAR_INPUT
		ipContainer	:	ITcVnContainer;	(* Container with TcVnVector3_INT elements, in which the element at position nIndex is replaced by aElement *)
		nIndex	:	ULINT;	(* Index *)
		hrPrev	:	HRESULT;	(* HRESULT indicating the result of previous operations (If SUCCEEDED(hrPrev) equals false, no operation is executed.) *)
	END_VAR

END_FUNCTION

// Functions/Basic Container Operations/F_VN_SetAt/F_VN_SetAt_TcVnVector3_REAL

	{attribute 'TcIecLibraryType'}
	{attribute 'external_name' := 'F_VN_SetAt_TcVnVector3_REAL_GUID_E7E10DE5_BBDC_D2B5_82C3_D03B676D1019'}
	(* Sets the element at the specified index of the container. *)
	FUNCTION F_VN_SetAt_TcVnVector3_REAL : HRESULT
	VAR_IN_OUT
		aElement	:	TcVnVector3_REAL;	(* Element to set at the specified container position *)
	END_VAR
	VAR_INPUT
		ipContainer	:	ITcVnContainer;	(* Container with TcVnVector3_REAL elements, in which the element at position nIndex is replaced by aElement *)
		nIndex	:	ULINT;	(* Index *)
		hrPrev	:	HRESULT;	(* HRESULT indicating the result of previous operations (If SUCCEEDED(hrPrev) equals false, no operation is executed.) *)
	END_VAR

END_FUNCTION

// Functions/Basic Container Operations/F_VN_SetAt/F_VN_SetAt_TcVnVector3_SINT

	{attribute 'TcIecLibraryType'}
	{attribute 'external_name' := 'F_VN_SetAt_TcVnVector3_SINT_GUID_F25AB548_5F5E_DC98_B6BC_12B5548547A2'}
	(* Sets the element at the specified index of the container. *)
	FUNCTION F_VN_SetAt_TcVnVector3_SINT : HRESULT
	VAR_IN_OUT
		aElement	:	TcVnVector3_SINT;	(* Element to set at the specified container position *)
	END_VAR
	VAR_INPUT
		ipContainer	:	ITcVnContainer;	(* Container with TcVnVector3_SINT elements, in which the element at position nIndex is replaced by aElement *)
		nIndex	:	ULINT;	(* Index *)
		hrPrev	:	HRESULT;	(* HRESULT indicating the result of previous operations (If SUCCEEDED(hrPrev) equals false, no operation is executed.) *)
	END_VAR

END_FUNCTION

// Functions/Basic Container Operations/F_VN_SetAt/F_VN_SetAt_TcVnVector3_UINT

	{attribute 'TcIecLibraryType'}
	{attribute 'external_name' := 'F_VN_SetAt_TcVnVector3_UINT_GUID_C0EAE934_C854_D169_9697_13D208B74332'}
	(* Sets the element at the specified index of the container. *)
	FUNCTION F_VN_SetAt_TcVnVector3_UINT : HRESULT
	VAR_IN_OUT
		aElement	:	TcVnVector3_UINT;	(* Element to set at the specified container position *)
	END_VAR
	VAR_INPUT
		ipContainer	:	ITcVnContainer;	(* Container with TcVnVector3_UINT elements, in which the element at position nIndex is replaced by aElement *)
		nIndex	:	ULINT;	(* Index *)
		hrPrev	:	HRESULT;	(* HRESULT indicating the result of previous operations (If SUCCEEDED(hrPrev) equals false, no operation is executed.) *)
	END_VAR

END_FUNCTION

// Functions/Basic Container Operations/F_VN_SetAt/F_VN_SetAt_TcVnVector3_USINT

	{attribute 'TcIecLibraryType'}
	{attribute 'external_name' := 'F_VN_SetAt_TcVnVector3_USINT_GUID_BA06F0BE_A1AF_D5B9_9020_C48B8FF58FCA'}
	(* Sets the element at the specified index of the container. *)
	FUNCTION F_VN_SetAt_TcVnVector3_USINT : HRESULT
	VAR_IN_OUT
		aElement	:	TcVnVector3_USINT;	(* Element to set at the specified container position *)
	END_VAR
	VAR_INPUT
		ipContainer	:	ITcVnContainer;	(* Container with TcVnVector3_USINT elements, in which the element at position nIndex is replaced by aElement *)
		nIndex	:	ULINT;	(* Index *)
		hrPrev	:	HRESULT;	(* HRESULT indicating the result of previous operations (If SUCCEEDED(hrPrev) equals false, no operation is executed.) *)
	END_VAR

END_FUNCTION

// Functions/Basic Container Operations/F_VN_SetAt/F_VN_SetAt_TcVnVector4_DINT

	{attribute 'TcIecLibraryType'}
	{attribute 'external_name' := 'F_VN_SetAt_TcVnVector4_DINT_GUID_F499B98D_2623_D67F_9D86_B597EF831028'}
	(* Sets the element at the specified index of the container. *)
	FUNCTION F_VN_SetAt_TcVnVector4_DINT : HRESULT
	VAR_IN_OUT
		aElement	:	TcVnVector4_DINT;	(* Element to set at the specified container position *)
	END_VAR
	VAR_INPUT
		ipContainer	:	ITcVnContainer;	(* Container with TcVnVector4_DINT elements, in which the element at position nIndex is replaced by aElement *)
		nIndex	:	ULINT;	(* Index *)
		hrPrev	:	HRESULT;	(* HRESULT indicating the result of previous operations (If SUCCEEDED(hrPrev) equals false, no operation is executed.) *)
	END_VAR

END_FUNCTION

// Functions/Basic Container Operations/F_VN_SetAt/F_VN_SetAt_TcVnVector4_INT

	{attribute 'TcIecLibraryType'}
	{attribute 'external_name' := 'F_VN_SetAt_TcVnVector4_INT_GUID_3C1822B1_48CA_DE5C_9E46_7B4DAA7D5C91'}
	(* Sets the element at the specified index of the container. *)
	FUNCTION F_VN_SetAt_TcVnVector4_INT : HRESULT
	VAR_IN_OUT
		aElement	:	TcVnVector4_INT;	(* Element to set at the specified container position *)
	END_VAR
	VAR_INPUT
		ipContainer	:	ITcVnContainer;	(* Container with TcVnVector4_INT elements, in which the element at position nIndex is replaced by aElement *)
		nIndex	:	ULINT;	(* Index *)
		hrPrev	:	HRESULT;	(* HRESULT indicating the result of previous operations (If SUCCEEDED(hrPrev) equals false, no operation is executed.) *)
	END_VAR

END_FUNCTION

// Functions/Basic Container Operations/F_VN_SetAt/F_VN_SetAt_TcVnVector4_LREAL

	{attribute 'TcIecLibraryType'}
	{attribute 'external_name' := 'F_VN_SetAt_TcVnVector4_LREAL_GUID_C31FA288_C1E2_DFBA_959D_2529D6A83E64'}
	(* Sets the element at the specified index of the container. *)
	FUNCTION F_VN_SetAt_TcVnVector4_LREAL : HRESULT
	VAR_IN_OUT
		aElement	:	TcVnVector4_LREAL;	(* Element to set at the specified container position *)
	END_VAR
	VAR_INPUT
		ipContainer	:	ITcVnContainer;	(* Container with TcVnVector4_LREAL elements, in which the element at position nIndex is replaced by aElement *)
		nIndex	:	ULINT;	(* Index *)
		hrPrev	:	HRESULT;	(* HRESULT indicating the result of previous operations (If SUCCEEDED(hrPrev) equals false, no operation is executed.) *)
	END_VAR

END_FUNCTION

// Functions/Basic Container Operations/F_VN_SetAt/F_VN_SetAt_TcVnVector4_REAL

	{attribute 'TcIecLibraryType'}
	{attribute 'external_name' := 'F_VN_SetAt_TcVnVector4_REAL_GUID_14303487_AE28_D413_B77E_42801EACBB76'}
	(* Sets the element at the specified index of the container. *)
	FUNCTION F_VN_SetAt_TcVnVector4_REAL : HRESULT
	VAR_IN_OUT
		aElement	:	TcVnVector4_REAL;	(* Element to set at the specified container position *)
	END_VAR
	VAR_INPUT
		ipContainer	:	ITcVnContainer;	(* Container with TcVnVector4_REAL elements, in which the element at position nIndex is replaced by aElement *)
		nIndex	:	ULINT;	(* Index *)
		hrPrev	:	HRESULT;	(* HRESULT indicating the result of previous operations (If SUCCEEDED(hrPrev) equals false, no operation is executed.) *)
	END_VAR

END_FUNCTION

// Functions/Basic Container Operations/F_VN_SetAt/F_VN_SetAt_TcVnVector4_SINT

	{attribute 'TcIecLibraryType'}
	{attribute 'external_name' := 'F_VN_SetAt_TcVnVector4_SINT_GUID_EABA744D_28BE_D87B_AF4B_7CA5F5619B72'}
	(* Sets the element at the specified index of the container. *)
	FUNCTION F_VN_SetAt_TcVnVector4_SINT : HRESULT
	VAR_IN_OUT
		aElement	:	TcVnVector4_SINT;	(* Element to set at the specified container position *)
	END_VAR
	VAR_INPUT
		ipContainer	:	ITcVnContainer;	(* Container with TcVnVector4_SINT elements, in which the element at position nIndex is replaced by aElement *)
		nIndex	:	ULINT;	(* Index *)
		hrPrev	:	HRESULT;	(* HRESULT indicating the result of previous operations (If SUCCEEDED(hrPrev) equals false, no operation is executed.) *)
	END_VAR

END_FUNCTION

// Functions/Basic Container Operations/F_VN_SetAt/F_VN_SetAt_TcVnVector4_UINT

	{attribute 'TcIecLibraryType'}
	{attribute 'external_name' := 'F_VN_SetAt_TcVnVector4_UINT_GUID_ECE2D899_7CF8_D3D2_B546_AEA5C3AC0E78'}
	(* Sets the element at the specified index of the container. *)
	FUNCTION F_VN_SetAt_TcVnVector4_UINT : HRESULT
	VAR_IN_OUT
		aElement	:	TcVnVector4_UINT;	(* Element to set at the specified container position *)
	END_VAR
	VAR_INPUT
		ipContainer	:	ITcVnContainer;	(* Container with TcVnVector4_UINT elements, in which the element at position nIndex is replaced by aElement *)
		nIndex	:	ULINT;	(* Index *)
		hrPrev	:	HRESULT;	(* HRESULT indicating the result of previous operations (If SUCCEEDED(hrPrev) equals false, no operation is executed.) *)
	END_VAR

END_FUNCTION

// Functions/Basic Container Operations/F_VN_SetAt/F_VN_SetAt_TcVnVector4_USINT

	{attribute 'TcIecLibraryType'}
	{attribute 'external_name' := 'F_VN_SetAt_TcVnVector4_USINT_GUID_FC552792_92A1_D187_8C56_50F5B0CDF203'}
	(* Sets the element at the specified index of the container. *)
	FUNCTION F_VN_SetAt_TcVnVector4_USINT : HRESULT
	VAR_IN_OUT
		aElement	:	TcVnVector4_USINT;	(* Element to set at the specified container position *)
	END_VAR
	VAR_INPUT
		ipContainer	:	ITcVnContainer;	(* Container with TcVnVector4_USINT elements, in which the element at position nIndex is replaced by aElement *)
		nIndex	:	ULINT;	(* Index *)
		hrPrev	:	HRESULT;	(* HRESULT indicating the result of previous operations (If SUCCEEDED(hrPrev) equals false, no operation is executed.) *)
	END_VAR

END_FUNCTION

// Functions/Basic Container Operations/F_VN_SetAt/F_VN_SetAt_UDINT

	{attribute 'TcIecLibraryType'}
	{attribute 'external_name' := 'F_VN_SetAt_UDINT_GUID_B305A6D1_2AE2_D412_9BD3_F3AF279AFF3A'}
	(* Sets the element at the specified index of the container. *)
	FUNCTION F_VN_SetAt_UDINT : HRESULT
	VAR_INPUT
		nElement	:	UDINT;	(* Element to set at the specified container position *)
		ipContainer	:	ITcVnContainer;	(* Container with UDINT elements, in which the element at position nIndex is replaced by nElement *)
		nIndex	:	ULINT;	(* Index *)
		hrPrev	:	HRESULT;	(* HRESULT indicating the result of previous operations (If SUCCEEDED(hrPrev) equals false, no operation is executed.) *)
	END_VAR

END_FUNCTION

// Functions/Basic Container Operations/F_VN_SetAt/F_VN_SetAt_UINT

	{attribute 'TcIecLibraryType'}
	{attribute 'external_name' := 'F_VN_SetAt_UINT_GUID_E7A3ED31_6DA7_DBE5_B80B_892891209441'}
	(* Sets the element at the specified index of the container. *)
	FUNCTION F_VN_SetAt_UINT : HRESULT
	VAR_INPUT
		nElement	:	UINT;	(* Element to set at the specified container position *)
		ipContainer	:	ITcVnContainer;	(* Container with UINT elements, in which the element at position nIndex is replaced by nElement *)
		nIndex	:	ULINT;	(* Index *)
		hrPrev	:	HRESULT;	(* HRESULT indicating the result of previous operations (If SUCCEEDED(hrPrev) equals false, no operation is executed.) *)
	END_VAR

END_FUNCTION

// Functions/Basic Container Operations/F_VN_SetAt/F_VN_SetAt_ULINT

	{attribute 'TcIecLibraryType'}
	{attribute 'external_name' := 'F_VN_SetAt_ULINT_GUID_8C16F2A2_3A38_D764_A670_EC92096893B4'}
	(* Sets the element at the specified index of the container. *)
	FUNCTION F_VN_SetAt_ULINT : HRESULT
	VAR_INPUT
		nElement	:	ULINT;	(* Element to set at the specified container position *)
		ipContainer	:	ITcVnContainer;	(* Container with ULINT elements, in which the element at position nIndex is replaced by nElement *)
		nIndex	:	ULINT;	(* Index *)
		hrPrev	:	HRESULT;	(* HRESULT indicating the result of previous operations (If SUCCEEDED(hrPrev) equals false, no operation is executed.) *)
	END_VAR

END_FUNCTION

// Functions/Basic Container Operations/F_VN_SetAt/F_VN_SetAt_USINT

	{attribute 'TcIecLibraryType'}
	{attribute 'external_name' := 'F_VN_SetAt_USINT_GUID_01F9B48C_F95B_D032_BABB_6175AD7802C9'}
	(* Sets the element at the specified index of the container. *)
	FUNCTION F_VN_SetAt_USINT : HRESULT
	VAR_INPUT
		nElement	:	USINT;	(* Element to set at the specified container position *)
		ipContainer	:	ITcVnContainer;	(* Container with USINT elements, in which the element at position nIndex is replaced by nElement *)
		nIndex	:	ULINT;	(* Index *)
		hrPrev	:	HRESULT;	(* HRESULT indicating the result of previous operations (If SUCCEEDED(hrPrev) equals false, no operation is executed.) *)
	END_VAR

END_FUNCTION

// Functions/Geometric and Coordinate Transformations/Calibration/F_VN_CalibrateCamera

	{attribute 'TcIecLibraryType'}
	{attribute 'external_name' := 'F_VN_CalibrateCamera_GUID_9B2FBB81_8252_DB75_B660_94F1805C04A3'}
	(* Compute the camera parameters (intrinsic + extrinsic) by evaluating an image containing a calibration pattern (circles). *)
	FUNCTION F_VN_CalibrateCamera : HRESULT
	VAR_INPUT
		ipSrcImage	:	ITcVnImage;	(* Source image containing a calibration pattern (1 channel, USINT elements) *)
		ipReferencePoints	:	ITcVnContainer;	(* Reference calibration pattern point positions (ContainerType_Vector_TcVnPoint3_REAL) *)
	END_VAR
	VAR_IN_OUT
		aCameraMatrix	:	TcVnMatrix3x3_LREAL;	(* Returns the camera matrix *)
		aDistortionCoefficients	:	TcVnArray8_LREAL;	(* Returns the lens distortion coefficients [k1, k2, p1, p2, k3, k4, k5, k6] *)
		aRotationMatrix	:	TcVnMatrix3x3_LREAL;	(* Returns the rotation matrix *)
		aTranslationVector	:	TcVnVector3_LREAL;	(* Returns the translation vector *)
		fReprojError	:	LREAL;	(* Returns the reprojection error *)
		stBlobDetectionParams	:	TcVnParamsBlobDetection;	(* Parameters for the internally used F_VN_DetectBlobs function *)
		stCalibrationOptions	:	TcVnCameraCalibrationOptions;	(* Calibration options *)
	END_VAR
	VAR_INPUT
		hrPrev	:	HRESULT;	(* HRESULT indicating the result of previous operations (If SUCCEEDED(hrPrev) equals false, no operation is executed.) *)
	END_VAR

END_FUNCTION

// Functions/Geometric and Coordinate Transformations/Calibration/F_VN_CalibrateCameraExp

	{attribute 'TcIecLibraryType'}
	{attribute 'external_name' := 'F_VN_CalibrateCameraExp_GUID_6DFA7B68_75C9_D42F_ADB8_B06E5FC95F85'}
	(* Compute the camera parameters (intrinsic + extrinsic) by evaluating images containing a calibration pattern (circles). The extrinsic parameters are computed for the first image in the array. (expert function) *)
	FUNCTION F_VN_CalibrateCameraExp : HRESULT
	VAR_INPUT
		pSrcImages	:	PVOID;	(* Pointer to an array of source images, each containing the same calibration pattern (1 channel, USINT elements) *)
		nSrcArraySize	:	UINT;	(* pSrcImages array size *)
		ipReferencePoints	:	ITcVnContainer;	(* Reference calibration pattern point positions (ContainerType_Vector_TcVnPoint3_REAL) *)
	END_VAR
	VAR_IN_OUT
		aCameraMatrix	:	TcVnMatrix3x3_LREAL;	(* Returns the camera matrix *)
		aDistortionCoefficients	:	TcVnArray8_LREAL;	(* Returns the lens distortion coefficients [k1, k2, p1, p2, k3, k4, k5, k6] *)
		aRotationMatrix	:	TcVnMatrix3x3_LREAL;	(* Returns the rotation matrix *)
		aTranslationVector	:	TcVnVector3_LREAL;	(* Returns the translation vector *)
		fReprojError	:	LREAL;	(* Returns the reprojection error *)
		stBlobDetectionParams	:	TcVnParamsBlobDetection;	(* Parameters for the internally used F_VN_DetectBlobs function *)
		stCalibrationOptions	:	TcVnCameraCalibrationOptions;	(* Calibration options *)
	END_VAR
	VAR_INPUT
		hrPrev	:	HRESULT;	(* HRESULT indicating the result of previous operations (If SUCCEEDED(hrPrev) equals false, no operation is executed.) *)
	END_VAR

END_FUNCTION

// Functions/Geometric and Coordinate Transformations/Calibration/F_VN_CalibrateCameraExp2

	{attribute 'TcIecLibraryType'}
	{attribute 'external_name' := 'F_VN_CalibrateCameraExp2_GUID_F91FD084_0889_D6C9_88FE_55F3E6C2586A'}
	(* Compute the camera parameters (intrinsic + extrinsic) by evaluating images containing a calibration pattern (circles). The extrinsic parameters are computed for the first image in the array. (expert function) *)
	FUNCTION F_VN_CalibrateCameraExp2 : HRESULT
	VAR_INPUT
		pSrcImages	:	PVOID;	(* Pointer to an array of source images, each containing the same calibration pattern (1 channel, USINT elements) *)
		nSrcArraySize	:	UINT;	(* pSrcImages array size *)
		ipReferencePoints	:	ITcVnContainer;	(* Reference calibration pattern point positions (ContainerType_Vector_TcVnPoint3_REAL) *)
	END_VAR
	VAR_IN_OUT
		aCameraMatrix	:	TcVnMatrix3x3_LREAL;	(* Returns the camera matrix *)
		aDistortionCoefficients	:	TcVnArray8_LREAL;	(* Returns the lens distortion coefficients [k1, k2, p1, p2, k3, k4, k5, k6] *)
		aRotationMatrix	:	TcVnMatrix3x3_LREAL;	(* Returns the rotation matrix *)
		aTranslationVector	:	TcVnVector3_LREAL;	(* Returns the translation vector *)
		fReprojError	:	LREAL;	(* Returns the reprojection error *)
		stBlobDetectionParams	:	TcVnParamsBlobDetection;	(* Parameters for the internally used F_VN_DetectBlobs function *)
		stCalibrationOptions	:	TcVnCameraCalibrationOptions;	(* Calibration options *)
	END_VAR
	VAR_INPUT
		bSubpixelAccuracy	:	BOOL;	(* If true, the pattern points are detected with subpixel accuracy *)
		eEdgeDirection	:	ETcVnEdgeDirection;	(* Specification of the edge direction to search for (from center to outside ellipse) *)
		fMinStrength	:	REAL;	(* Specification of the minimum strength (intensity difference) of the edge to search for *)
		nMaxThickness	:	UDINT;	(* Specification of the maximum thickness of the edge to search for, which means fMinStrength must be reached within nMaxThickness pixels *)
		nSubpixelsIterations	:	UDINT;	(* Specifies the number of subpixels (for INTERPOLATION, 10 - 20 usually is sufficient) or maximum number of iterations for optimizing the parameters (for APPROX_ERF and APPROX_GAUSSIAN, 50 - 100 usually is sufficient) *)
		nSearchLines	:	UDINT;	(* Specifies the amount of search lines, which are equally distributed in all directions (must be >= 8 and a multiple of 4) *)
		fApproxPrecision	:	REAL;	(* Specifies the approximation precision for APPROX_ERF and APPROX_GAUSSIAN (0.001 usually is sufficient, unused for INTERPOLATION) *)
		eAlgorithm	:	ETcVnEdgeDetectionAlgorithm;	(* Selection of the edge detection algorithm *)
		hrPrev	:	HRESULT;	(* HRESULT indicating the result of previous operations (If SUCCEEDED(hrPrev) equals false, no operation is executed.) *)
	END_VAR

END_FUNCTION

// Functions/Geometric and Coordinate Transformations/Calibration/F_VN_CalibrateCameraExp3

	{attribute 'TcIecLibraryType'}
	{attribute 'external_name' := 'F_VN_CalibrateCameraExp3_GUID_A96D25D5_EAC8_D8B8_A480_F9AD7844ABC0'}
	(* Compute the camera parameters (intrinsic + extrinsic) by evaluating images containing a calibration pattern (circles). The extrinsic parameters are computed for the first image in the array. (expert function) *)
	FUNCTION F_VN_CalibrateCameraExp3 : HRESULT
	VAR_INPUT
		pSrcImages	:	PVOID;	(* Pointer to an array of source images, each containing the same calibration pattern (1 channel, USINT elements) *)
		nSrcArraySize	:	UINT;	(* pSrcImages array size *)
		ipReferencePoints	:	ITcVnContainer;	(* Reference calibration pattern point positions (ContainerType_Vector_TcVnPoint3_REAL) *)
	END_VAR
	VAR_IN_OUT
		aCameraMatrix	:	TcVnMatrix3x3_LREAL;	(* Returns the camera matrix *)
		aDistortionCoefficients	:	TcVnArray8_LREAL;	(* Returns the lens distortion coefficients [k1, k2, p1, p2, k3, k4, k5, k6] *)
		aRotationMatrix	:	TcVnMatrix3x3_LREAL;	(* Returns the rotation matrix *)
		aTranslationVector	:	TcVnVector3_LREAL;	(* Returns the translation vector *)
		fReprojError	:	LREAL;	(* Returns the reprojection error *)
		stBlobDetectionParams	:	TcVnParamsBlobDetection;	(* Parameters for the internally used F_VN_DetectBlobs function *)
		stCalibrationOptions	:	TcVnCameraCalibrationOptions;	(* Calibration options *)
	END_VAR
	VAR_INPUT
		bSubpixelAccuracy	:	BOOL;	(* If true, the pattern points are detected with subpixel accuracy *)
		eEdgeDirection	:	ETcVnEdgeDirection;	(* Specification of the edge direction to search for (from center to outside ellipse) *)
		fMinStrength	:	REAL;	(* Specification of the minimum strength (intensity difference) of the edge to search for *)
		nMaxThickness	:	UDINT;	(* Specification of the maximum thickness of the edge to search for, which means fMinStrength must be reached within nMaxThickness pixels *)
		nSubpixelsIterations	:	UDINT;	(* Specifies the number of subpixels (for INTERPOLATION, 10 - 20 usually is sufficient) or maximum number of iterations for optimizing the parameters (for APPROX_ERF and APPROX_GAUSSIAN, 50 - 100 usually is sufficient) *)
		nSearchLines	:	UDINT;	(* Specifies the amount of search lines, which are equally distributed in all directions (must be >= 8 and a multiple of 4) *)
		fApproxPrecision	:	REAL;	(* Specifies the approximation precision for APPROX_ERF and APPROX_GAUSSIAN (0.001 usually is sufficient, unused for INTERPOLATION) *)
		eAlgorithm	:	ETcVnEdgeDetectionAlgorithm;	(* Selection of the edge detection algorithm *)
		eWorldSystem	:	ETcVnWorldCoordinateSystem;	(* World coordinate system orientation *)
		hrPrev	:	HRESULT;	(* HRESULT indicating the result of previous operations (If SUCCEEDED(hrPrev) equals false, no operation is executed.) *)
	END_VAR

END_FUNCTION

// Functions/Geometric and Coordinate Transformations/Calibration/F_VN_CalibrateCameraManually

	{attribute 'TcIecLibraryType'}
	{attribute 'external_name' := 'F_VN_CalibrateCameraManually_GUID_2D3DE9EE_C246_DFD2_B1D8_E74798503039'}
	(* Compute the camera parameters (intrinsic + extrinsic). The extrinsic parameters are computed for the first inner container. *)
	FUNCTION F_VN_CalibrateCameraManually : HRESULT
	VAR_INPUT
		ipImagePoints	:	ITcVnContainer;	(* Provided image points of multiple images (ContainerType_Vector_Vector_TcVnPoint2_REAL, each inner container with at least 6 points). The container and point order must match ipReferencePoints. *)
		nImageWidth	:	UDINT;	(* Image width *)
		nImageHeight	:	UDINT;	(* Image height *)
		ipReferencePoints	:	ITcVnContainer;	(* Reference world points (ContainerType_Vector_Vector_TcVnPoint3_REAL). The number of inner containers and their amount of points must match ipImagePoints. *)
	END_VAR
	VAR_IN_OUT
		aCameraMatrix	:	TcVnMatrix3x3_LREAL;	(* Returns the camera matrix *)
		aDistortionCoefficients	:	TcVnArray8_LREAL;	(* Returns the lens distortion coefficients [k1, k2, p1, p2, k3, k4, k5, k6] *)
		aRotationMatrix	:	TcVnMatrix3x3_LREAL;	(* Returns the rotation matrix (for the first inner container) *)
		aTranslationVector	:	TcVnVector3_LREAL;	(* Returns the translation vector (for the first inner container) *)
		fReprojError	:	LREAL;	(* Returns the reprojection error *)
		stCalibrationOptions	:	TcVnCameraCalibrationOptions;	(* Calibration options *)
	END_VAR
	VAR_INPUT
		hrPrev	:	HRESULT;	(* HRESULT indicating the result of previous operations (If SUCCEEDED(hrPrev) equals false, no operation is executed.) *)
	END_VAR

END_FUNCTION

// Functions/Geometric and Coordinate Transformations/Calibration/F_VN_CalibrateCameraManuallyExp

	{attribute 'TcIecLibraryType'}
	{attribute 'external_name' := 'F_VN_CalibrateCameraManuallyExp_GUID_AE53830D_70E7_D6F8_BDF3_9107182054EB'}
	(* Compute the camera parameters (intrinsic + extrinsic). The extrinsic parameters are computed for the first inner container. (expert function) *)
	FUNCTION F_VN_CalibrateCameraManuallyExp : HRESULT
	VAR_INPUT
		ipImagePoints	:	ITcVnContainer;	(* Provided image points of multiple images (ContainerType_Vector_Vector_TcVnPoint2_REAL, each inner container with at least 6 points). The container and point order must match ipReferencePoints. *)
		nImageWidth	:	UDINT;	(* Image width *)
		nImageHeight	:	UDINT;	(* Image height *)
		ipReferencePoints	:	ITcVnContainer;	(* Reference world points (ContainerType_Vector_Vector_TcVnPoint3_REAL). The number of inner containers and their amount of points must match ipImagePoints. *)
	END_VAR
	VAR_IN_OUT
		aCameraMatrix	:	TcVnMatrix3x3_LREAL;	(* Returns the camera matrix *)
		aDistortionCoefficients	:	TcVnArray8_LREAL;	(* Returns the lens distortion coefficients [k1, k2, p1, p2, k3, k4, k5, k6] *)
		aRotationMatrix	:	TcVnMatrix3x3_LREAL;	(* Returns the rotation matrix (for the first inner container) *)
		aTranslationVector	:	TcVnVector3_LREAL;	(* Returns the translation vector (for the first inner container) *)
		fReprojError	:	LREAL;	(* Returns the reprojection error *)
		stCalibrationOptions	:	TcVnCameraCalibrationOptions;	(* Calibration options *)
	END_VAR
	VAR_INPUT
		eWorldSystem	:	ETcVnWorldCoordinateSystem;	(* World coordinate system orientation *)
		hrPrev	:	HRESULT;	(* HRESULT indicating the result of previous operations (If SUCCEEDED(hrPrev) equals false, no operation is executed.) *)
	END_VAR

END_FUNCTION

// Functions/Geometric and Coordinate Transformations/Calibration/F_VN_CalibrateCameraPlanar

	{attribute 'TcIecLibraryType'}
	{attribute 'external_name' := 'F_VN_CalibrateCameraPlanar_GUID_AD13E504_55B8_D1FB_9908_AC4EDA179941'}
	(* Calibrate camera using a planar calibration pattern comprised of four circles marking the corners of a rectangle. *)
	FUNCTION F_VN_CalibrateCameraPlanar : HRESULT
	VAR_INPUT
		ipSrcImage	:	ITcVnImage;	(* Binary source image (background zero, markers non-zero) *)
	END_VAR
	VAR_IN_OUT
		aMarkerPositions	:	TcVnArray4_Point2_REAL;	(* Marker positions within their plane using world units (right-handed coordinate system) *)
		aTransformationMatrix	:	TcVnMatrix3x3_LREAL;	(* Returns a 3-by-3 matrix for the transformation from image coordinates into the reference coordinate system *)
	END_VAR
	VAR_INPUT
		hrPrev	:	HRESULT;	(* HRESULT indicating the result of previous operations (If SUCCEEDED(hrPrev) equals false, no operation is executed.) *)
	END_VAR

END_FUNCTION

// Functions/Geometric and Coordinate Transformations/Calibration/F_VN_CalibrateCameraPlanarExp

	{attribute 'TcIecLibraryType'}
	{attribute 'external_name' := 'F_VN_CalibrateCameraPlanarExp_GUID_0D7431C6_9AE2_DCFC_8CDE_41A9F22D51F9'}
	(* Calibrate camera using a planar calibration pattern comprised of four circles marking the corners of a rectangle. (expert function) *)
	FUNCTION F_VN_CalibrateCameraPlanarExp : HRESULT
	VAR_INPUT
		ipSrcImage	:	ITcVnImage;	(* Binary source image (background zero, markers non-zero) *)
	END_VAR
	VAR_IN_OUT
		aMarkerPositions	:	TcVnArray4_Point2_REAL;	(* Marker positions within their plane using world units (right-handed coordinate system) *)
		aTransformationMatrix	:	TcVnMatrix3x3_LREAL;	(* Returns a 3-by-3 matrix for the transformation from image coordinates into the reference coordinate system *)
		aMarkerImagePositions	:	TcVnArray4_Point2_REAL;	(* Returns the marker positions in image coordinates (left-handed coordinate system) *)
	END_VAR
	VAR_INPUT
		nMinMarkerArea	:	UDINT;	(* Minimum area for the detection of markers (Smaller markers are ignored.) *)
		nMaxMarkerArea	:	UDINT;	(* Maximum area for the detection of markers (Larger markers are ignored.) *)
		fMaxMarkerEccentricity	:	LREAL;	(* Maximum eccenticity for the detection of markers (The eccentricity measures deviations from a round shape (eccentricity = 0: round object; eccentricity = 1.0:  linear object).) *)
		hrPrev	:	HRESULT;	(* HRESULT indicating the result of previous operations (If SUCCEEDED(hrPrev) equals false, no operation is executed.) *)
	END_VAR

END_FUNCTION

// Functions/Geometric and Coordinate Transformations/Calibration/F_VN_CalibrateLinescanCamera

	{attribute 'TcIecLibraryType'}
	{attribute 'external_name' := 'F_VN_CalibrateLinescanCamera_GUID_F0955690_9DB6_DC5B_92AA_2F2839F09C5C'}
	(* Compute the camera parameters (intrinsic + extrinsic) by evaluating images containing a line calibration pattern. The pattern must consist of alternating vertical and diagonal lines, with each diagonal having the same constant slope: |\|\|...\|. The results are only valid for the x-direction of a line scan image. To get accurate x-values for a transformation into world coordinates, the y-coordinate must be set to half the sensor width and so equal to the cy-value of the camera matrix. For other y-values, the results are approximated and can be inaccurate. The extrinsic parameters are computed for the first image in the array. *)
	FUNCTION F_VN_CalibrateLinescanCamera : HRESULT
	VAR_INPUT
		pSrcImages	:	PVOID;	(* Pointer to an array of 1 or more source images (1 channel). If the images have more than 1 row, each row must contain an image of the same pattern position. *)
		nSrcArraySize	:	UINT;	(* pSrcImages array size *)
		ipPatternLineOrigins	:	ITcVnContainer;	(* X position of the pattern line origins (ContainerType_Vector_REAL, usually same origin for vertical and following diagonal line) *)
		fSlopeRad	:	LREAL;	(* Slope of the diagonal line in rad (> 0, < PI/2), relative to the vertical line (i.e., 0 would be a vertical line, PI/2 a horizontal line) *)
	END_VAR
	VAR_IN_OUT
		aCameraMatrix	:	TcVnMatrix3x3_LREAL;	(* Returns the camera matrix *)
		aDistortionCoefficients	:	TcVnArray8_LREAL;	(* Returns the lens distortion coefficients [k1, k2, p1, p2, k3, k4, k5, k6] *)
		aRotationMatrix	:	TcVnMatrix3x3_LREAL;	(* Returns the rotation matrix *)
		aTranslationVector	:	TcVnVector3_LREAL;	(* Returns the translation vector *)
		fReprojError	:	LREAL;	(* Returns the reprojection error *)
		stCalibrationOptions	:	TcVnCameraCalibrationOptions;	(* Calibration options (recommended to set bFixAspectRatio, bFixPrincipalPoint, bZeroTangentDist) *)
	END_VAR
	VAR_INPUT
		eEdgeDirection	:	ETcVnEdgeDirection;	(* Specification of the edge direction to search for *)
		hrPrev	:	HRESULT;	(* HRESULT indicating the result of previous operations (If SUCCEEDED(hrPrev) equals false, no operation is executed.) *)
	END_VAR

END_FUNCTION

// Functions/Geometric and Coordinate Transformations/Calibration/F_VN_CalibrateLinescanCameraExp

	{attribute 'TcIecLibraryType'}
	{attribute 'external_name' := 'F_VN_CalibrateLinescanCameraExp_GUID_DDF9FD17_ABFC_D988_BA19_C6282829533D'}
	(* Compute the camera parameters (intrinsic + extrinsic) by evaluating images containing a line calibration pattern. The pattern must consist of alternating vertical and diagonal lines, with each diagonal having the same constant slope: |\|\|...\|. The results are only valid for the x-direction of a line scan image. To get accurate x-values for a transformation into world coordinates, the y-coordinate must be set to half the sensor width and so equal to the cy-value of the camera matrix. For other y-values, the results are approximated and can be inaccurate. The extrinsic parameters are computed for the first image in the array. (expert function) *)
	FUNCTION F_VN_CalibrateLinescanCameraExp : HRESULT
	VAR_INPUT
		pSrcImages	:	PVOID;	(* Pointer to an array of 1 or more source images (1 channel). If the images have more than 1 row, each row must contain an image of the same pattern position. *)
		nSrcArraySize	:	UINT;	(* pSrcImages array size *)
		ipPatternLineOrigins	:	ITcVnContainer;	(* X position of the pattern line origins (ContainerType_Vector_REAL, usually same origin for vertical and following diagonal line) *)
		fSlopeRad	:	LREAL;	(* Slope of the diagonal line in rad (> 0, < PI/2), relative to the vertical line (i.e., 0 would be a vertical line, PI/2 a horizontal line) *)
	END_VAR
	VAR_IN_OUT
		aCameraMatrix	:	TcVnMatrix3x3_LREAL;	(* Returns the camera matrix *)
		aDistortionCoefficients	:	TcVnArray8_LREAL;	(* Returns the lens distortion coefficients [k1, k2, p1, p2, k3, k4, k5, k6] *)
		aRotationMatrix	:	TcVnMatrix3x3_LREAL;	(* Returns the rotation matrix *)
		aTranslationVector	:	TcVnVector3_LREAL;	(* Returns the translation vector *)
		fReprojError	:	LREAL;	(* Returns the reprojection error *)
		stCalibrationOptions	:	TcVnCameraCalibrationOptions;	(* Calibration options (recommended to set bFixAspectRatio, bFixPrincipalPoint, bZeroTangentDist) *)
	END_VAR
	VAR_INPUT
		eEdgeDirection	:	ETcVnEdgeDirection;	(* Specification of the edge direction to search for *)
		fMinStrength	:	REAL;	(* Specification of the minimum strength (intensity difference) of the edge to search for *)
		nMaxSearchLines	:	UDINT;	(* Maximum number of search lines (equally distributed over the image height, at most 1 searchline per image row) *)
		nMaxThickness	:	UDINT;	(* Specification of the maximum thickness of the edge to search for, which means fMinStrength must be reached within nMaxThickness pixels *)
		nSubpixelsIterations	:	UDINT;	(* Specifies the number of subpixels (for INTERPOLATION, 10 - 20 usually is sufficient) or maximum number of iterations for optimizing the parameters (for APPROX_ERF and APPROX_GAUSSIAN, 50 - 100 usually is sufficient) *)
		fApproxPrecision	:	REAL;	(* Specifies the approximation precision for APPROX_ERF and APPROX_GAUSSIAN (0.001 usually is sufficient, unused for INTERPOLATION) *)
		eAlgorithm	:	ETcVnEdgeDetectionAlgorithm;	(* Selection of the edge detection algorithm *)
		hrPrev	:	HRESULT;	(* HRESULT indicating the result of previous operations (If SUCCEEDED(hrPrev) equals false, no operation is executed.) *)
	END_VAR

END_FUNCTION

// Functions/Geometric and Coordinate Transformations/Calibration/F_VN_CompensateLensDistortion

	{attribute 'TcIecLibraryType'}
	{attribute 'external_name' := 'F_VN_CompensateLensDistortion_GUID_38041498_CF3F_D2E2_A530_6CF25178D498'}
	(* Transforms an image to compensate the lens distortion. *)
	FUNCTION F_VN_CompensateLensDistortion : HRESULT
	VAR_INPUT
		ipSrcImage	:	ITcVnImage;	(* Source image *)
		ipDestImage	:	REFERENCE TO ITcVnImage;	(* Destination image (An appropriate destination image will be created if required.) *)
	END_VAR
	VAR_IN_OUT
		aCameraMatrix	:	TcVnMatrix3x3_LREAL;	(* Camera matrix containing the intrinsic parameters *)
		aDistortionCoefficients	:	TcVnArray4_LREAL;	(* Lens distortion coefficients [k1, k2, p1, p2] *)
	END_VAR
	VAR_INPUT
		hrPrev	:	HRESULT;	(* HRESULT indicating the result of previous operations (If SUCCEEDED(hrPrev) equals false, no operation is executed.) *)
	END_VAR

END_FUNCTION

// Functions/Geometric and Coordinate Transformations/Calibration/F_VN_CompensateLensDistortionExp1

	{attribute 'TcIecLibraryType'}
	{attribute 'external_name' := 'F_VN_CompensateLensDistortionExp1_GUID_A279729F_931C_DEF9_A2A4_7B371020E818'}
	(* Transforms an image to compensate the lens distortion. (expert function) *)
	FUNCTION F_VN_CompensateLensDistortionExp1 : HRESULT
	VAR_INPUT
		ipSrcImage	:	ITcVnImage;	(* Source image *)
		ipDestImage	:	REFERENCE TO ITcVnImage;	(* Destination image (An appropriate destination image will be created if required.) *)
	END_VAR
	VAR_IN_OUT
		aCameraMatrix	:	TcVnMatrix3x3_LREAL;	(* Camera matrix containing the intrinsic parameters *)
		aDistortionCoefficients	:	TcVnArray8_LREAL;	(* Lens distortion coefficients [k1, k2, p1, p2, k3, k4, k5, k6] *)
	END_VAR
	VAR_INPUT
		hrPrev	:	HRESULT;	(* HRESULT indicating the result of previous operations (If SUCCEEDED(hrPrev) equals false, no operation is executed.) *)
	END_VAR

END_FUNCTION

// Functions/Geometric and Coordinate Transformations/Calibration/F_VN_CompensateLensDistortionExp2

	{attribute 'TcIecLibraryType'}
	{attribute 'external_name' := 'F_VN_CompensateLensDistortionExp2_GUID_5DE22D13_D619_DEFB_86A0_D4306D891468'}
	(* Transforms an image to compensate the lens distortion. (expert function) *)
	FUNCTION F_VN_CompensateLensDistortionExp2 : HRESULT
	VAR_INPUT
		ipSrcImage	:	ITcVnImage;	(* Source image *)
		ipDestImage	:	REFERENCE TO ITcVnImage;	(* Destination image (An appropriate destination image will be created if required.) *)
	END_VAR
	VAR_IN_OUT
		aCameraMatrix	:	TcVnMatrix3x3_LREAL;	(* Camera matrix containing the intrinsic parameters *)
		aDistortionCoefficients	:	TcVnArray8_LREAL;	(* Lens distortion coefficients [k1, k2, p1, p2, k3, k4, k5, k6] *)
		aNewCameraMatrix	:	TcVnMatrix3x3_LREAL;	(* Allows additional scaling and shifting of the result image *)
	END_VAR
	VAR_INPUT
		hrPrev	:	HRESULT;	(* HRESULT indicating the result of previous operations (If SUCCEEDED(hrPrev) equals false, no operation is executed.) *)
	END_VAR

END_FUNCTION

// Functions/Geometric and Coordinate Transformations/Calibration/F_VN_CompensateLensDistortionForPoints

	{attribute 'TcIecLibraryType'}
	{attribute 'external_name' := 'F_VN_CompensateLensDistortionForPoints_GUID_859CAFF4_28B5_DECF_9E81_FB25B0F02B02'}
	(* Transforms point coordinates to compensate the lens distortion. *)
	FUNCTION F_VN_CompensateLensDistortionForPoints : HRESULT
	VAR_INPUT
		ipSrcPoints	:	ITcVnContainer;	(* Container with source point coordinates (ContainerType_Vector_TcVnPoint2_REAL or ContainerType_Vector_TcVnPoint2_DINT) *)
		ipDestPoints	:	REFERENCE TO ITcVnContainer;	(* Returns a container with the transformed point coordinates (ContainerType_Vector_TcVnPoint2_REAL) *)
	END_VAR
	VAR_IN_OUT
		aCameraMatrix	:	TcVnMatrix3x3_LREAL;	(* Camera matrix containing the intrinsic parameters *)
		aDistortionCoefficients	:	TcVnArray4_LREAL;	(* Lens distortion coefficients [k1, k2, p1, p2] *)
	END_VAR
	VAR_INPUT
		hrPrev	:	HRESULT;	(* HRESULT indicating the result of previous operations (If SUCCEEDED(hrPrev) equals false, no operation is executed.) *)
	END_VAR

END_FUNCTION

// Functions/Geometric and Coordinate Transformations/Calibration/F_VN_CompensateLensDistortionForPointsExp1

	{attribute 'TcIecLibraryType'}
	{attribute 'external_name' := 'F_VN_CompensateLensDistortionForPointsExp1_GUID_E4697840_2B82_DEE7_AFA3_D4BC69E1808C'}
	(* Transforms point coordinates to compensate the lens distortion. (expert function) *)
	FUNCTION F_VN_CompensateLensDistortionForPointsExp1 : HRESULT
	VAR_INPUT
		ipSrcPoints	:	ITcVnContainer;	(* Container with source point coordinates (ContainerType_Vector_TcVnPoint2_REAL or ContainerType_Vector_TcVnPoint2_DINT) *)
		ipDestPoints	:	REFERENCE TO ITcVnContainer;	(* Returns a container with the transformed point coordinates (ContainerType_Vector_TcVnPoint2_REAL) *)
	END_VAR
	VAR_IN_OUT
		aCameraMatrix	:	TcVnMatrix3x3_LREAL;	(* Camera matrix containing the intrinsic parameters *)
		aDistortionCoefficients	:	TcVnArray8_LREAL;	(* Lens distortion coefficients [k1, k2, p1, p2, k3, k4, k5, k6] *)
	END_VAR
	VAR_INPUT
		hrPrev	:	HRESULT;	(* HRESULT indicating the result of previous operations (If SUCCEEDED(hrPrev) equals false, no operation is executed.) *)
	END_VAR

END_FUNCTION

// Functions/Geometric and Coordinate Transformations/Calibration/F_VN_CompensateLensDistortionForPointsExp2

	{attribute 'TcIecLibraryType'}
	{attribute 'external_name' := 'F_VN_CompensateLensDistortionForPointsExp2_GUID_ABB82CAF_9EF5_D4D3_8D27_5A1A89CE7159'}
	(* Transforms point coordinates to compensate the lens distortion. (expert function) *)
	FUNCTION F_VN_CompensateLensDistortionForPointsExp2 : HRESULT
	VAR_INPUT
		ipSrcPoints	:	ITcVnContainer;	(* Container with source point coordinates (ContainerType_Vector_TcVnPoint2_REAL or ContainerType_Vector_TcVnPoint2_DINT) *)
		ipDestPoints	:	REFERENCE TO ITcVnContainer;	(* Returns a container with the transformed point coordinates (ContainerType_Vector_TcVnPoint2_REAL) *)
	END_VAR
	VAR_IN_OUT
		aCameraMatrix	:	TcVnMatrix3x3_LREAL;	(* Camera matrix containing the intrinsic parameters *)
		aDistortionCoefficients	:	TcVnArray8_LREAL;	(* Lens distortion coefficients [k1, k2, p1, p2, k3, k4, k5, k6] *)
		aNewCameraMatrix	:	TcVnMatrix3x3_LREAL;	(* Allows additional shifting of the result point coordinates *)
	END_VAR
	VAR_INPUT
		hrPrev	:	HRESULT;	(* HRESULT indicating the result of previous operations (If SUCCEEDED(hrPrev) equals false, no operation is executed.) *)
	END_VAR

END_FUNCTION

// Functions/Geometric and Coordinate Transformations/Calibration/F_VN_DetectPatternPoints

	{attribute 'TcIecLibraryType'}
	{attribute 'external_name' := 'F_VN_DetectPatternPoints_GUID_7E575849_FA25_D875_8150_47B690AFDD6E'}
	(* Detects calibration pattern points (circles) within the provided image. *)
	FUNCTION F_VN_DetectPatternPoints : HRESULT
	VAR_INPUT
		ipSrcImage	:	ITcVnImage;	(* Source image (USINT, 1 channel) *)
		ipPatternPoints	:	REFERENCE TO ITcVnContainer;	(* Returns the pattern point positions (ContainerType_Vector_TcVnPoint2_REAL; Non-zero interface pointers are reused.) *)
	END_VAR
	VAR_IN_OUT
		stBlobDetectionParams	:	TcVnParamsBlobDetection;	(* Parameters to detect and filter contours. *)
	END_VAR
	VAR_INPUT
		nNumberOfPoints	:	UDINT;	(* Expected number of pattern points *)
		hrPrev	:	HRESULT;	(* HRESULT indicating the result of previous operations (If SUCCEEDED(hrPrev) equals false, no operation is executed.) *)
	END_VAR

END_FUNCTION

// Functions/Geometric and Coordinate Transformations/Calibration/F_VN_DetectPatternPointsExp

	{attribute 'TcIecLibraryType'}
	{attribute 'external_name' := 'F_VN_DetectPatternPointsExp_GUID_903823F9_9D6B_D624_9699_5FCAC0D5F886'}
	(* Detects calibration pattern points (circles) within the provided image. (expert function) *)
	FUNCTION F_VN_DetectPatternPointsExp : HRESULT
	VAR_INPUT
		ipSrcImage	:	ITcVnImage;	(* Source image (USINT, 1 channel) *)
		ipPatternPoints	:	REFERENCE TO ITcVnContainer;	(* Returns the pattern point positions (ContainerType_Vector_TcVnPoint2_REAL; Non-zero interface pointers are reused.) *)
	END_VAR
	VAR_IN_OUT
		stBlobDetectionParams	:	TcVnParamsBlobDetection;	(* Parameters to detect and filter contours. *)
	END_VAR
	VAR_INPUT
		nNumberOfPoints	:	UDINT;	(* Expected number of pattern points *)
		fSizeDiffThresFactor	:	REAL;	(* Threshold for filtering contours by average size *)
		bSubpixelAccuracy	:	BOOL;	(* If true, the pattern points are detected with subpixel accuracy *)
		eEdgeDirection	:	ETcVnEdgeDirection;	(* Specification of the edge direction to search for (from center to outside circle) *)
		fMinStrength	:	REAL;	(* Specification of the minimum strength (intensity difference) of the edge to search for *)
		nMaxThickness	:	UDINT;	(* Specification of the maximum thickness of the edge to search for, which means fMinStrength must be reached within nMaxThickness pixels *)
		nSubpixelsIterations	:	UDINT;	(* Specifies the number of subpixels (for INTERPOLATION, 10 - 20 usually is sufficient) or maximum number of iterations for optimizing the parameters (for APPROX_ERF and APPROX_GAUSSIAN, 50 - 100 usually is sufficient) *)
		nSearchLines	:	UDINT;	(* Specifies the amount of search lines, which are equally distributed in all directions (must be >= 8 and a multiple of 4) *)
		fApproxPrecision	:	REAL;	(* Specifies the approximation precision for APPROX_ERF and APPROX_GAUSSIAN (0.001 usually is sufficient, unused for INTERPOLATION) *)
		eAlgorithm	:	ETcVnEdgeDetectionAlgorithm;	(* Selection of the edge detection algorithm *)
		hrPrev	:	HRESULT;	(* HRESULT indicating the result of previous operations (If SUCCEEDED(hrPrev) equals false, no operation is executed.) *)
	END_VAR

END_FUNCTION

// Functions/Geometric and Coordinate Transformations/Calibration/F_VN_GenerateCalibrationPatternReferencePoints

	{attribute 'TcIecLibraryType'}
	{attribute 'external_name' := 'F_VN_GenerateCalibrationPatternReferencePoints_GUID_C67720A1_4192_D3E3_8ADB_2A5AD64EDF2F'}
	(* Generate reference points for common calibration patterns. *)
	FUNCTION F_VN_GenerateCalibrationPatternReferencePoints : HRESULT
	VAR_INPUT
		ipReferencePoints	:	REFERENCE TO ITcVnContainer;	(* Returns the generated reference points (ContainerType_Vector_TcVnPoint3_REAL) *)
		ePattern	:	ETcVnCalibrationPattern;	(* Calibration pattern type *)
		eOrigin	:	ETcVnCalibrationPatternOrigin;	(* Calibration pattern origin *)
		nWidth	:	UDINT;	(* Pattern width, i.e. number of pattern points in x direction *)
		nHeight	:	UDINT;	(* Pattern height, i.e. number of pattern points in y direction *)
		fDistX	:	REAL;	(* Distance between pattern points in x direction *)
		fDistY	:	REAL;	(* Distance between pattern points in y direction *)
		hrPrev	:	HRESULT;	(* HRESULT indicating the result of previous operations (If SUCCEEDED(hrPrev) equals false, no operation is executed.) *)
	END_VAR

END_FUNCTION

// Functions/Geometric and Coordinate Transformations/Calibration/F_VN_ImagePointsWorldDistance

	{attribute 'TcIecLibraryType'}
	{attribute 'external_name' := 'F_VN_ImagePointsWorldDistance_GUID_98B59F88_610B_DF11_BEC6_8E3FD932D074'}
	(* Computes the distance in the world coordinate system between two points (in the same world coordinate z layer) given in image coordinates. *)
	FUNCTION F_VN_ImagePointsWorldDistance : HRESULT
	VAR_IN_OUT
		aImagePoint1	:	TcVnPoint2_REAL;	(* First point in the image coordinate system *)
		aImagePoint2	:	TcVnPoint2_REAL;	(* Second point in the image coordinate system *)
		fWorldDistance	:	LREAL;	(* Returns the distance between aImagePoint1 and aImagePoint2 in the world coordinate system *)
		aCameraMatrix	:	TcVnMatrix3x3_LREAL;	(* 3x3 camera matrix containing the intrinsic parameters *)
		aDistortionCoefficients	:	TcVnArray8_LREAL;	(* Lens distortion coefficients [k1, k2, p1, p2, k3, k4, k5, k6] *)
		aRotationMatrix	:	TcVnMatrix3x3_LREAL;	(* 3x3 rotation matrix *)
		aTranslationVector	:	TcVnVector3_LREAL;	(* Translation vector *)
	END_VAR
	VAR_INPUT
		fZ	:	LREAL;	(* z coordinate (world coordinate system) of the given points (0 would be at (toplevel) calibration pattern) *)
		hrPrev	:	HRESULT;	(* HRESULT indicating the result of previous operations (If SUCCEEDED(hrPrev) equals false, no operation is executed.) *)
	END_VAR

END_FUNCTION

// Functions/Geometric and Coordinate Transformations/Calibration/F_VN_SolvePnP

	{attribute 'TcIecLibraryType'}
	{attribute 'external_name' := 'F_VN_SolvePnP_GUID_D33356AC_E80D_D153_B8C7_419D93A346C6'}
	(* Computes the rotation matrix and translation vector from 3D-2D point correspondences. *)
	FUNCTION F_VN_SolvePnP : HRESULT
	VAR_INPUT
		ipImagePoints	:	ITcVnContainer;	(* Image points (ContainerType_Vector_TcVnPoint2_REAL, requires at least 4 points in the same order as in ipReferencePoints) *)
		ipReferencePoints	:	ITcVnContainer;	(* Reference world points (ContainerType_Vector_TcVnPoint3_REAL, same number of points as in ipImagePoints) *)
	END_VAR
	VAR_IN_OUT
		aCameraMatrix	:	TcVnMatrix3x3_LREAL;	(* Camera matrix (e.g. computed with one of the CalibrateCamera functions) *)
		aDistortionCoefficients	:	TcVnArray8_LREAL;	(* Lens distortion coefficients [k1, k2, p1, p2, k3, k4, k5, k6] (e.g. computed with one of the CalibrateCamera functions) *)
		aRotationMatrix	:	TcVnMatrix3x3_LREAL;	(* Returns the rotation matrix *)
		aTranslationVector	:	TcVnVector3_LREAL;	(* Returns the translation vector *)
		fReprojError	:	LREAL;	(* Returns the reprojection error *)
	END_VAR
	VAR_INPUT
		hrPrev	:	HRESULT;	(* HRESULT indicating the result of previous operations (If SUCCEEDED(hrPrev) equals false, no operation is executed.) *)
	END_VAR

END_FUNCTION

// Functions/Geometric and Coordinate Transformations/Calibration/F_VN_SolvePnPExp

	{attribute 'TcIecLibraryType'}
	{attribute 'external_name' := 'F_VN_SolvePnPExp_GUID_D1EA1655_61CC_D324_96D9_450DC65AC741'}
	(* Computes the rotation matrix and translation vector from 3D-2D point correspondences. (expert function) *)
	FUNCTION F_VN_SolvePnPExp : HRESULT
	VAR_INPUT
		ipImagePoints	:	ITcVnContainer;	(* Image points (ContainerType_Vector_TcVnPoint2_REAL, requires at least 4 points in the same order as in ipReferencePoints) *)
		ipReferencePoints	:	ITcVnContainer;	(* Reference world points (ContainerType_Vector_TcVnPoint3_REAL, same number of points as in ipImagePoints) *)
	END_VAR
	VAR_IN_OUT
		aCameraMatrix	:	TcVnMatrix3x3_LREAL;	(* Camera matrix (e.g. computed with one of the CalibrateCamera functions) *)
		aDistortionCoefficients	:	TcVnArray8_LREAL;	(* Lens distortion coefficients [k1, k2, p1, p2, k3, k4, k5, k6] (e.g. computed with one of the CalibrateCamera functions) *)
		aRotationMatrix	:	TcVnMatrix3x3_LREAL;	(* Returns the rotation matrix *)
		aTranslationVector	:	TcVnVector3_LREAL;	(* Returns the translation vector *)
		fReprojError	:	LREAL;	(* Returns the reprojection error *)
	END_VAR
	VAR_INPUT
		eMethod	:	ETcVnSolvePnPMethod;	(* Solve PnP method *)
		bUseExtrinsicGuess	:	BOOL;	(* If true, the provided rotation matrix and translation vector are used as an initial guess for further optimization (only supported for the SPM_ITERATIVE method). *)
		hrPrev	:	HRESULT;	(* HRESULT indicating the result of previous operations (If SUCCEEDED(hrPrev) equals false, no operation is executed.) *)
	END_VAR

END_FUNCTION

// Functions/Geometric and Coordinate Transformations/Calibration/F_VN_SortDetectedPatternPoints

	{attribute 'TcIecLibraryType'}
	{attribute 'external_name' := 'F_VN_SortDetectedPatternPoints_GUID_3AFE2BCB_3495_D09D_9328_6835C3F09855'}
	(* Sort the detected pattern points according to the relative positions of the calibration pattern points. *)
	FUNCTION F_VN_SortDetectedPatternPoints : HRESULT
	VAR_INPUT
		ipImagePoints	:	ITcVnContainer;	(* Detected pattern point positions in the image coordinate system (will be sorted by this function, ContainerType_Vector_TcVnPoint2_REAL) *)
		ipPatternPoints	:	ITcVnContainer;	(* The pattern points in the calibration pattern coordinate system, used as a reference to sort ipImagePoints (ContainerType_Vector_TcVnPoint3_REAL) *)
		hrPrev	:	HRESULT;	(* HRESULT indicating the result of previous operations (If SUCCEEDED(hrPrev) equals false, no operation is executed.) *)
	END_VAR

END_FUNCTION

// Functions/Geometric and Coordinate Transformations/Calibration/F_VN_TransformCoordinatesPlanar_Container

	{attribute 'TcIecLibraryType'}
	{attribute 'external_name' := 'F_VN_TransformCoordinatesPlanar_Container_GUID_F8B93D0A_49F5_D59E_BE8A_B89D5B7F4DCD'}
	(* Compute real-world coordinates for given image points or vice versa. *)
	FUNCTION F_VN_TransformCoordinatesPlanar_Container : HRESULT
	VAR_INPUT
		ipSrcPoints	:	ITcVnContainer;	(* Container with 2D source points (TcVnPoint2_DINT or TcVnPoint2_REAL or TcVnPoint2_LREAL) *)
		ipDestPoints	:	REFERENCE TO ITcVnContainer;	(* Returns the transformed 2D points (TcVnPoint2_LREAL) *)
	END_VAR
	VAR_IN_OUT
		aTransformationMatrix	:	TcVnMatrix3x3_LREAL;	(* Transformation matrix obtained with VnCalibrateCameraPlanar() or its inverse matrix obtained with VnInvertMatrix3x3() *)
	END_VAR
	VAR_INPUT
		hrPrev	:	HRESULT;	(* HRESULT indicating the result of previous operations (If SUCCEEDED(hrPrev) equals false, no operation is executed.) *)
	END_VAR

END_FUNCTION

// Functions/Geometric and Coordinate Transformations/Calibration/F_VN_TransformCoordinatesPlanar_Point

	{attribute 'TcIecLibraryType'}
	{attribute 'external_name' := 'F_VN_TransformCoordinatesPlanar_Point_GUID_0C438016_6606_D674_B056_690F6F20CC37'}
	(* Compute real-world coordinates for a given image point or vice versa. *)
	FUNCTION F_VN_TransformCoordinatesPlanar_Point : HRESULT
	VAR_IN_OUT
		aSrcPoint	:	TcVnPoint2_LREAL;	(* Point in the source coordinate system *)
		aDestPoint	:	TcVnPoint2_LREAL;	(* Returns point in the destination coordinate system *)
		aTransformationMatrix	:	TcVnMatrix3x3_LREAL;	(* Transformation matrix obtained with VnCalibrateCameraPlanar() or its inverse matrix obtained with VnInvertMatrix3x3() *)
	END_VAR
	VAR_INPUT
		hrPrev	:	HRESULT;	(* HRESULT indicating the result of previous operations (If SUCCEEDED(hrPrev) equals false, no operation is executed.) *)
	END_VAR

END_FUNCTION

// Functions/Geometric and Coordinate Transformations/Calibration/F_VN_TransformCoordinatesImageToWorld_Container

	{attribute 'TcIecLibraryType'}
	{attribute 'external_name' := 'F_VN_TransformCoordinatesImageToWorld_Container_GUID_CB2E98FF_3D83_D43B_81A0_70C8A286BF87'}
	(* Transform 2D image point coordinates to 3D world coordinates (using intrinsic + extrinsic calibration results). *)
	FUNCTION F_VN_TransformCoordinatesImageToWorld_Container : HRESULT
	VAR_INPUT
		ipSrcPoints2D	:	ITcVnContainer;	(* Container with 2D source points (TcVnPoint2_DINT or TcVnPoint2_REAL or TcVnPoint2_LREAL) *)
		ipDestPoints3D	:	REFERENCE TO ITcVnContainer;	(* Returns the transformed 3D points (TcVnPoint3_LREAL) *)
	END_VAR
	VAR_IN_OUT
		aCameraMatrix	:	TcVnMatrix3x3_LREAL;	(* 3x3 camera matrix containing the intrinsic parameters *)
		aDistortionCoefficients	:	TcVnArray8_LREAL;	(* Lens distortion coefficients [k1, k2, p1, p2, k3, k4, k5, k6] *)
		aRotationMatrix	:	TcVnMatrix3x3_LREAL;	(* 3x3 rotation matrix *)
		aTranslationVector	:	TcVnVector3_LREAL;	(* Translation vector *)
	END_VAR
	VAR_INPUT
		fZ	:	LREAL;	(* z coordinate (world coordinate system) of the transformed points (0 would be at (toplevel) calibration pattern) *)
		hrPrev	:	HRESULT;	(* HRESULT indicating the result of previous operations (If SUCCEEDED(hrPrev) equals false, no operation is executed.) *)
	END_VAR

END_FUNCTION

// Functions/Geometric and Coordinate Transformations/Calibration/F_VN_TransformCoordinatesImageToWorld_Point

	{attribute 'TcIecLibraryType'}
	{attribute 'external_name' := 'F_VN_TransformCoordinatesImageToWorld_Point_GUID_1C0C7109_0970_D5FF_B74D_615C2D58D2D9'}
	(* Transform 2D image point coordinate to 3D world coordinate (using intrinsic + extrinsic calibration results). *)
	FUNCTION F_VN_TransformCoordinatesImageToWorld_Point : HRESULT
	VAR_IN_OUT
		aSrcPoint	:	TcVnPoint2_LREAL;	(* Point in the image coordinate system *)
		aDestPoint	:	TcVnPoint3_LREAL;	(* Returns the point in the world coordinate system *)
		aCameraMatrix	:	TcVnMatrix3x3_LREAL;	(* 3x3 camera matrix containing the intrinsic parameters *)
		aDistortionCoefficients	:	TcVnArray8_LREAL;	(* Lens distortion coefficients [k1, k2, p1, p2, k3, k4, k5, k6] *)
		aRotationMatrix	:	TcVnMatrix3x3_LREAL;	(* 3x3 rotation matrix *)
		aTranslationVector	:	TcVnVector3_LREAL;	(* Translation vector *)
	END_VAR
	VAR_INPUT
		fZ	:	LREAL;	(* z coordinate (world coordinate system) of the transformed points (0 would be at (toplevel) calibration pattern) *)
		hrPrev	:	HRESULT;	(* HRESULT indicating the result of previous operations (If SUCCEEDED(hrPrev) equals false, no operation is executed.) *)
	END_VAR

END_FUNCTION

// Functions/Geometric and Coordinate Transformations/Calibration/F_VN_TransformCoordinatesWorldToImage_Container

	{attribute 'TcIecLibraryType'}
	{attribute 'external_name' := 'F_VN_TransformCoordinatesWorldToImage_Container_GUID_593885FB_2683_DBB7_B7DC_CFF51DF753A7'}
	(* Transform 3D world coordinates to 2D image coordinates (using intrinsic + extrinsic calibration results). *)
	FUNCTION F_VN_TransformCoordinatesWorldToImage_Container : HRESULT
	VAR_INPUT
		ipSrcPoints3D	:	ITcVnContainer;	(* Container with 3D source points (TcVnPoint3_LREAL) *)
		ipDestPoints2D	:	REFERENCE TO ITcVnContainer;	(* Returns the transformed 2D points (TcVnPoint2_REAL or TcVnPoint2_DINT, depending on bInteger) *)
	END_VAR
	VAR_IN_OUT
		aCameraMatrix	:	TcVnMatrix3x3_LREAL;	(* 3x3 camera matrix containing the intrinsic parameters *)
		aDistortionCoefficients	:	TcVnArray8_LREAL;	(* Lens distortion coefficients [k1, k2, p1, p2, k3, k4, k5, k6] *)
		aRotationMatrix	:	TcVnMatrix3x3_LREAL;	(* 3x3 rotation matrix *)
		aTranslationVector	:	TcVnVector3_LREAL;	(* Translation vector *)
	END_VAR
	VAR_INPUT
		bInteger	:	BOOL;	(* Selects whether the function returns a container of TcVnPoint2_DINT or TcVnPoint2_REAL *)
		hrPrev	:	HRESULT;	(* HRESULT indicating the result of previous operations (If SUCCEEDED(hrPrev) equals false, no operation is executed.) *)
	END_VAR

END_FUNCTION

// Functions/Geometric and Coordinate Transformations/Calibration/F_VN_TransformCoordinatesWorldToImage_Point

	{attribute 'TcIecLibraryType'}
	{attribute 'external_name' := 'F_VN_TransformCoordinatesWorldToImage_Point_GUID_1D0AECDB_0567_D0D5_B583_3EAB5DD4D7A9'}
	(* Transform 3D world coordinates to 2D image coordinates (using intrinsic + extrinsic calibration results). *)
	FUNCTION F_VN_TransformCoordinatesWorldToImage_Point : HRESULT
	VAR_IN_OUT
		aSrcPoint	:	TcVnPoint3_LREAL;	(* 3D source point (world coordinate system) *)
		aDestPoint	:	TcVnPoint2_REAL;	(* Returns the transformed 2D point (image coordinate system) *)
		aCameraMatrix	:	TcVnMatrix3x3_LREAL;	(* 3x3 camera matrix containing the intrinsic parameters *)
		aDistortionCoefficients	:	TcVnArray8_LREAL;	(* Lens distortion coefficients [k1, k2, p1, p2, k3, k4, k5, k6] *)
		aRotationMatrix	:	TcVnMatrix3x3_LREAL;	(* 3x3 rotation matrix *)
		aTranslationVector	:	TcVnVector3_LREAL;	(* Translation vector *)
	END_VAR
	VAR_INPUT
		hrPrev	:	HRESULT;	(* HRESULT indicating the result of previous operations (If SUCCEEDED(hrPrev) equals false, no operation is executed.) *)
	END_VAR

END_FUNCTION

// Functions/Container Statistics/F_VN_MaxElementElementwise/F_VN_MaxElementElementwise_DINT

	{attribute 'TcIecLibraryType'}
	{attribute 'external_name' := 'F_VN_MaxElementElementwise_DINT_GUID_3A3F03FA_EB12_DE3A_8F11_230DD4B9A00F'}
	(* Gets the element wise maximum container element. *)
	FUNCTION F_VN_MaxElementElementwise_DINT : HRESULT
	VAR_INPUT
		ipContainer	:	ITcVnContainer;	(* Source container *)
	END_VAR
	VAR_IN_OUT
		nMax	:	DINT;	(* Returns the requested element *)
	END_VAR
	VAR_INPUT
		hrPrev	:	HRESULT;	(* HRESULT indicating the result of previous operations (If SUCCEEDED(hrPrev) equals false, no operation is executed.) *)
	END_VAR

END_FUNCTION

// Functions/Container Statistics/F_VN_MaxElementElementwise/F_VN_MaxElementElementwise_INT

	{attribute 'TcIecLibraryType'}
	{attribute 'external_name' := 'F_VN_MaxElementElementwise_INT_GUID_0E368E4D_5ED1_DD91_B4F4_63F5ED1BD2DF'}
	(* Gets the element wise maximum container element. *)
	FUNCTION F_VN_MaxElementElementwise_INT : HRESULT
	VAR_INPUT
		ipContainer	:	ITcVnContainer;	(* Source container *)
	END_VAR
	VAR_IN_OUT
		nMax	:	INT;	(* Returns the requested element *)
	END_VAR
	VAR_INPUT
		hrPrev	:	HRESULT;	(* HRESULT indicating the result of previous operations (If SUCCEEDED(hrPrev) equals false, no operation is executed.) *)
	END_VAR

END_FUNCTION

// Functions/Container Statistics/F_VN_MaxElementElementwise/F_VN_MaxElementElementwise_LREAL

	{attribute 'TcIecLibraryType'}
	{attribute 'external_name' := 'F_VN_MaxElementElementwise_LREAL_GUID_D98B7A99_4CF6_D156_B567_A2BA431370A1'}
	(* Gets the element wise maximum container element. *)
	FUNCTION F_VN_MaxElementElementwise_LREAL : HRESULT
	VAR_INPUT
		ipContainer	:	ITcVnContainer;	(* Source container *)
	END_VAR
	VAR_IN_OUT
		fMax	:	LREAL;	(* Returns the requested element *)
	END_VAR
	VAR_INPUT
		hrPrev	:	HRESULT;	(* HRESULT indicating the result of previous operations (If SUCCEEDED(hrPrev) equals false, no operation is executed.) *)
	END_VAR

END_FUNCTION

// Functions/Container Statistics/F_VN_MaxElementElementwise/F_VN_MaxElementElementwise_REAL

	{attribute 'TcIecLibraryType'}
	{attribute 'external_name' := 'F_VN_MaxElementElementwise_REAL_GUID_B27ACE6C_D897_DC75_B867_4909C23EAA2F'}
	(* Gets the element wise maximum container element. *)
	FUNCTION F_VN_MaxElementElementwise_REAL : HRESULT
	VAR_INPUT
		ipContainer	:	ITcVnContainer;	(* Source container *)
	END_VAR
	VAR_IN_OUT
		fMax	:	REAL;	(* Returns the requested element *)
	END_VAR
	VAR_INPUT
		hrPrev	:	HRESULT;	(* HRESULT indicating the result of previous operations (If SUCCEEDED(hrPrev) equals false, no operation is executed.) *)
	END_VAR

END_FUNCTION

// Functions/Container Statistics/F_VN_MaxElementElementwise/F_VN_MaxElementElementwise_SINT

	{attribute 'TcIecLibraryType'}
	{attribute 'external_name' := 'F_VN_MaxElementElementwise_SINT_GUID_4CEBE539_04A5_D379_9F44_048545939BD5'}
	(* Gets the element wise maximum container element. *)
	FUNCTION F_VN_MaxElementElementwise_SINT : HRESULT
	VAR_INPUT
		ipContainer	:	ITcVnContainer;	(* Source container *)
	END_VAR
	VAR_IN_OUT
		nMax	:	SINT;	(* Returns the requested element *)
	END_VAR
	VAR_INPUT
		hrPrev	:	HRESULT;	(* HRESULT indicating the result of previous operations (If SUCCEEDED(hrPrev) equals false, no operation is executed.) *)
	END_VAR

END_FUNCTION

// Functions/Container Statistics/F_VN_MaxElementElementwise/F_VN_MaxElementElementwise_TcVnPoint2_DINT

	{attribute 'TcIecLibraryType'}
	{attribute 'external_name' := 'F_VN_MaxElementElementwise_TcVnPoint2_DINT_GUID_300C0963_CF55_DF7B_AD42_EB278FF8AD0C'}
	(* Gets the element wise maximum container element. *)
	FUNCTION F_VN_MaxElementElementwise_TcVnPoint2_DINT : HRESULT
	VAR_INPUT
		ipContainer	:	ITcVnContainer;	(* Source container *)
	END_VAR
	VAR_IN_OUT
		aMax	:	TcVnPoint2_DINT;	(* Returns the requested element *)
	END_VAR
	VAR_INPUT
		hrPrev	:	HRESULT;	(* HRESULT indicating the result of previous operations (If SUCCEEDED(hrPrev) equals false, no operation is executed.) *)
	END_VAR

END_FUNCTION

// Functions/Container Statistics/F_VN_MaxElementElementwise/F_VN_MaxElementElementwise_TcVnPoint2_LREAL

	{attribute 'TcIecLibraryType'}
	{attribute 'external_name' := 'F_VN_MaxElementElementwise_TcVnPoint2_LREAL_GUID_3E6C444F_8396_DFEA_8834_4D936AE628BC'}
	(* Gets the element wise maximum container element. *)
	FUNCTION F_VN_MaxElementElementwise_TcVnPoint2_LREAL : HRESULT
	VAR_INPUT
		ipContainer	:	ITcVnContainer;	(* Source container *)
	END_VAR
	VAR_IN_OUT
		aMax	:	TcVnPoint2_LREAL;	(* Returns the requested element *)
	END_VAR
	VAR_INPUT
		hrPrev	:	HRESULT;	(* HRESULT indicating the result of previous operations (If SUCCEEDED(hrPrev) equals false, no operation is executed.) *)
	END_VAR

END_FUNCTION

// Functions/Container Statistics/F_VN_MaxElementElementwise/F_VN_MaxElementElementwise_TcVnPoint2_REAL

	{attribute 'TcIecLibraryType'}
	{attribute 'external_name' := 'F_VN_MaxElementElementwise_TcVnPoint2_REAL_GUID_95954649_54E8_DC8E_AABE_2E41F77B6428'}
	(* Gets the element wise maximum container element. *)
	FUNCTION F_VN_MaxElementElementwise_TcVnPoint2_REAL : HRESULT
	VAR_INPUT
		ipContainer	:	ITcVnContainer;	(* Source container *)
	END_VAR
	VAR_IN_OUT
		aMax	:	TcVnPoint2_REAL;	(* Returns the requested element *)
	END_VAR
	VAR_INPUT
		hrPrev	:	HRESULT;	(* HRESULT indicating the result of previous operations (If SUCCEEDED(hrPrev) equals false, no operation is executed.) *)
	END_VAR

END_FUNCTION

// Functions/Container Statistics/F_VN_MaxElementElementwise/F_VN_MaxElementElementwise_TcVnPoint3_LREAL

	{attribute 'TcIecLibraryType'}
	{attribute 'external_name' := 'F_VN_MaxElementElementwise_TcVnPoint3_LREAL_GUID_91C02391_E227_D293_89FE_DD3C96E0C28E'}
	(* Gets the element wise maximum container element. *)
	FUNCTION F_VN_MaxElementElementwise_TcVnPoint3_LREAL : HRESULT
	VAR_INPUT
		ipContainer	:	ITcVnContainer;	(* Source container *)
	END_VAR
	VAR_IN_OUT
		aMax	:	TcVnPoint3_LREAL;	(* Returns the requested element *)
	END_VAR
	VAR_INPUT
		hrPrev	:	HRESULT;	(* HRESULT indicating the result of previous operations (If SUCCEEDED(hrPrev) equals false, no operation is executed.) *)
	END_VAR

END_FUNCTION

// Functions/Container Statistics/F_VN_MaxElementElementwise/F_VN_MaxElementElementwise_TcVnPoint3_REAL

	{attribute 'TcIecLibraryType'}
	{attribute 'external_name' := 'F_VN_MaxElementElementwise_TcVnPoint3_REAL_GUID_661D3463_7521_D33F_8ED5_FD427F245343'}
	(* Gets the element wise maximum container element. *)
	FUNCTION F_VN_MaxElementElementwise_TcVnPoint3_REAL : HRESULT
	VAR_INPUT
		ipContainer	:	ITcVnContainer;	(* Source container *)
	END_VAR
	VAR_IN_OUT
		aMax	:	TcVnPoint3_REAL;	(* Returns the requested element *)
	END_VAR
	VAR_INPUT
		hrPrev	:	HRESULT;	(* HRESULT indicating the result of previous operations (If SUCCEEDED(hrPrev) equals false, no operation is executed.) *)
	END_VAR

END_FUNCTION

// Functions/Container Statistics/F_VN_MaxElementElementwise/F_VN_MaxElementElementwise_TcVnVector2_DINT

	{attribute 'TcIecLibraryType'}
	{attribute 'external_name' := 'F_VN_MaxElementElementwise_TcVnVector2_DINT_GUID_5863BF52_1879_D574_9E62_0426E109BCC6'}
	(* Gets the element wise maximum container element. *)
	FUNCTION F_VN_MaxElementElementwise_TcVnVector2_DINT : HRESULT
	VAR_INPUT
		ipContainer	:	ITcVnContainer;	(* Source container *)
	END_VAR
	VAR_IN_OUT
		aMax	:	TcVnVector2_DINT;	(* Returns the requested element *)
	END_VAR
	VAR_INPUT
		hrPrev	:	HRESULT;	(* HRESULT indicating the result of previous operations (If SUCCEEDED(hrPrev) equals false, no operation is executed.) *)
	END_VAR

END_FUNCTION

